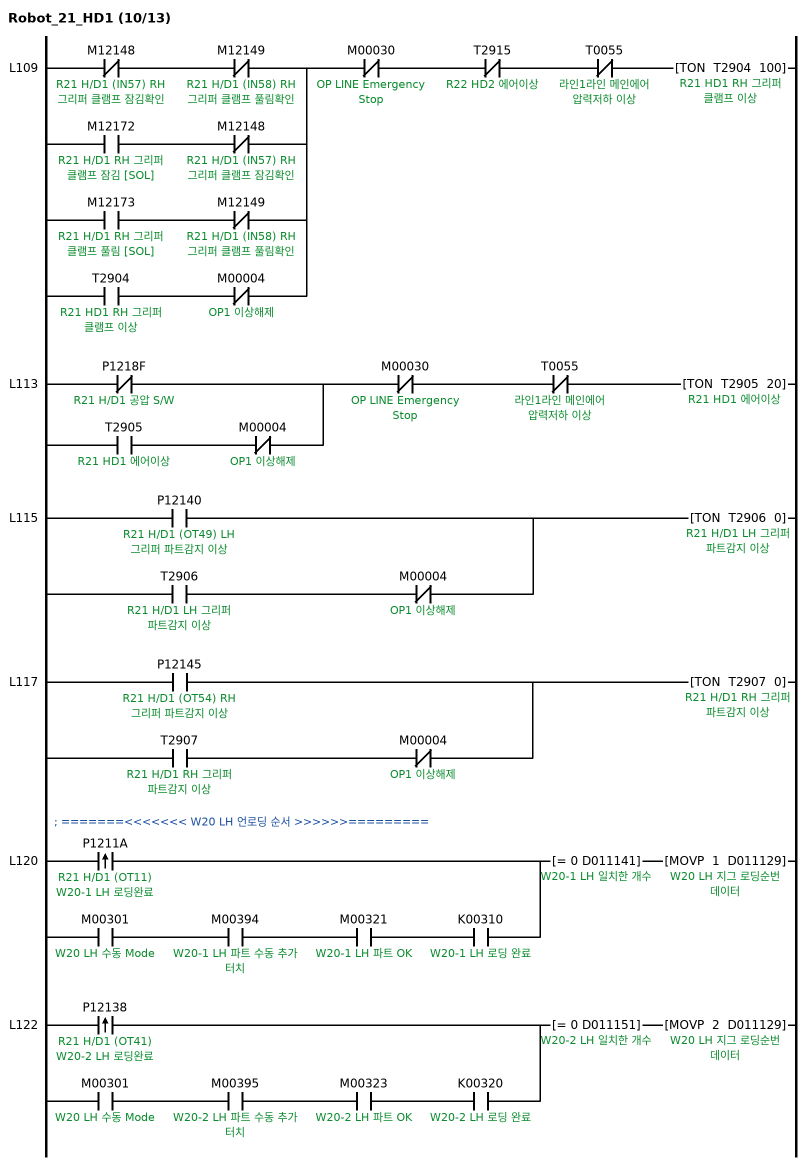
[picture p360: Robot_21_HD1 rungs L109-L122]
; L109
LOAD NOT  M12148	// R21 H/D1 (IN57) RH 그리퍼 클램프 잠김확인
AND NOT   M12149	// R21 H/D1 (IN58) RH 그리퍼 클램프 풀림확인
LOAD      M12172	// R21 H/D1 RH 그리퍼 클램프 잠김 [SOL]
AND NOT   M12148	// R21 H/D1 (IN57) RH 그리퍼 클램프 잠김확인
OR LOAD
LOAD      M12173	// R21 H/D1 RH 그리퍼 클램프 풀림 [SOL]
AND NOT   M12149	// R21 H/D1 (IN58) RH 그리퍼 클램프 풀림확인
OR LOAD
LOAD      T2904	// R21 HD1 RH 그리퍼 클램프 이상
AND NOT   M00004	// OP1 이상해제
OR LOAD
AND NOT   M00030	// OP LINE Emergency Stop
AND NOT   T2915	// R22 HD2 에어이상
AND NOT   T0055	// 라인1라인 메인에어 압력저하 이상
TON       T2904 100	// R21 HD1 RH 그리퍼 클램프 이상
; L113
LOAD NOT  P1218F	// R21 H/D1 공압 S/W
LOAD      T2905	// R21 HD1 에어이상
AND NOT   M00004	// OP1 이상해제
OR LOAD
AND NOT   M00030	// OP LINE Emergency Stop
AND NOT   T0055	// 라인1라인 메인에어 압력저하 이상
TON       T2905 20	// R21 HD1 에어이상
; L115
LOAD      P12140	// R21 H/D1 (OT49) LH 그리퍼 파트감지 이상
LOAD      T2906	// R21 H/D1 LH 그리퍼 파트감지 이상
AND NOT   M00004	// OP1 이상해제
OR LOAD
TON       T2906 0	// R21 H/D1 LH 그리퍼 파트감지 이상
; L117
LOAD      P12145	// R21 H/D1 (OT54) RH 그리퍼 파트감지 이상
LOAD      T2907	// R21 H/D1 RH 그리퍼 파트감지 이상
AND NOT   M00004	// OP1 이상해제
OR LOAD
TON       T2907 0	// R21 H/D1 RH 그리퍼 파트감지 이상
// =======<<<<<<< W20 LH 언로딩 순서 >>>>>>=========
; L120
LOADP     P1211A	// R21 H/D1 (OT11) W20-1 LH 로딩완료
LOAD      M00301	// W20 LH 수동 Mode
AND       M00394	// W20-1 LH 파트 수동 추가 터치
AND       M00321	// W20-1 LH 파트 OK
AND       K00310	// W20-1 LH 로딩 완료
OR LOAD
AND=      0 D011141	// W20-1 LH 일치한 개수
MOVP      1 D011129	// W20 LH 지그 로딩순번 데이터
; L122
LOADP     P12138	// R21 H/D1 (OT41) W20-2 LH 로딩완료
LOAD      M00301	// W20 LH 수동 Mode
AND       M00395	// W20-2 LH 파트 수동 추가 터치
AND       M00323	// W20-2 LH 파트 OK
AND       K00320	// W20-2 LH 로딩 완료
OR LOAD
AND=      0 D011151	// W20-2 LH 일치한 개수
MOVP      2 D011129	// W20 LH 지그 로딩순번 데이터

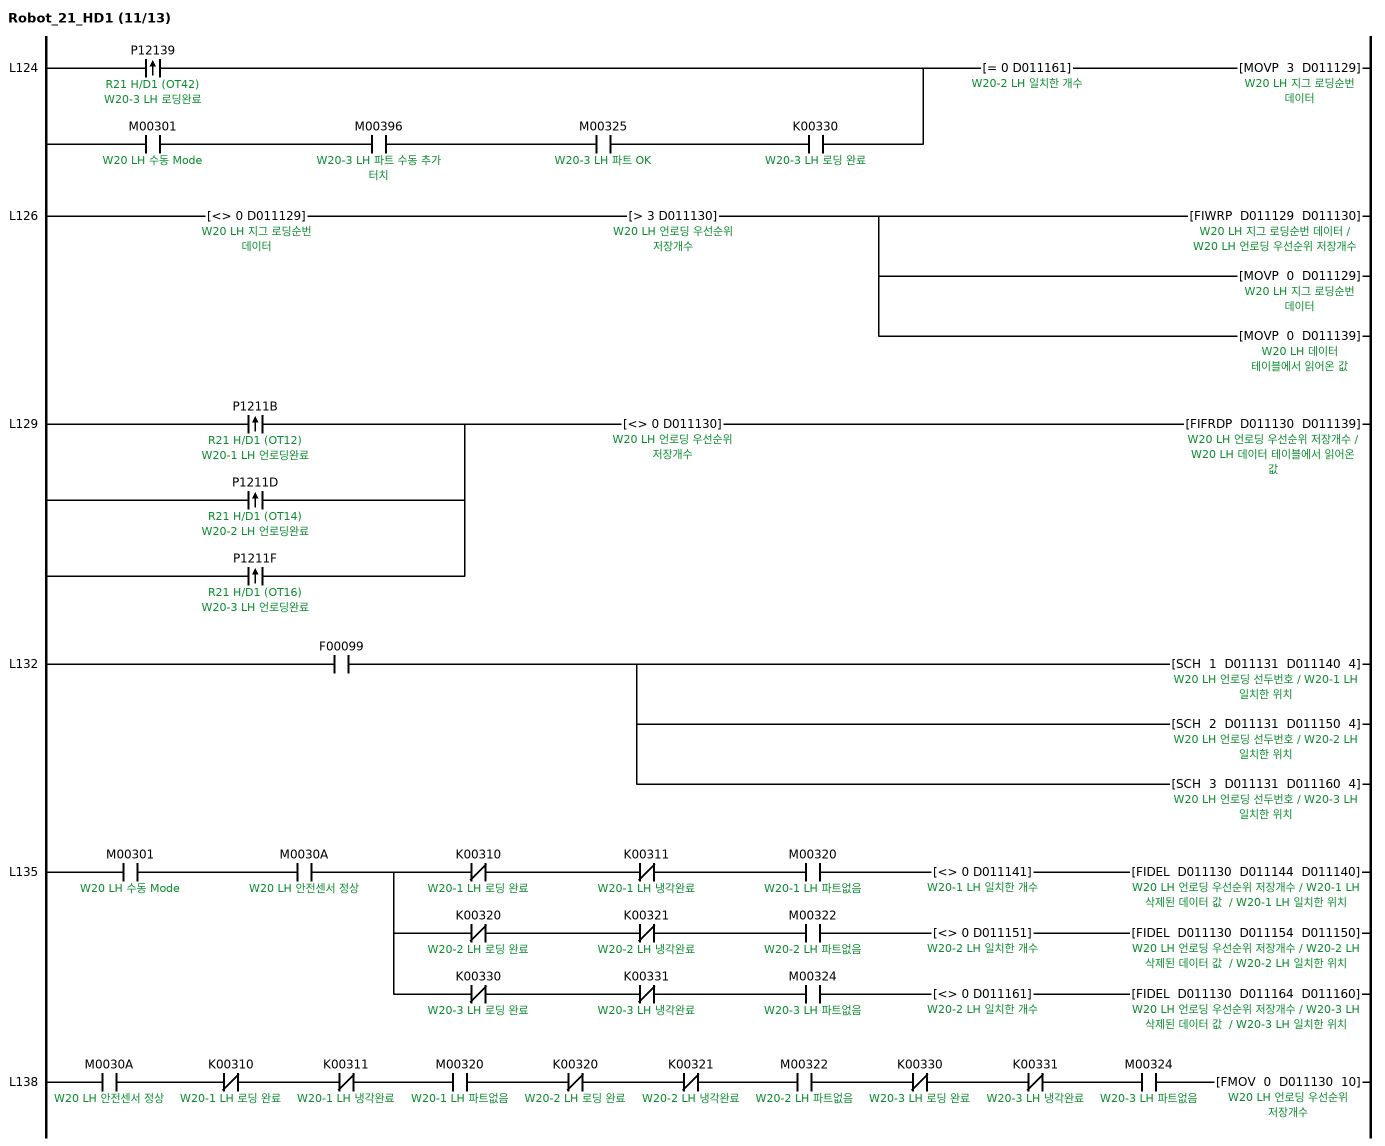
; L124
LOADP     P12139	// R21 H/D1 (OT42) W20-3 LH 로딩완료
LOAD      M00301	// W20 LH 수동 Mode
AND       M00396	// W20-3 LH 파트 수동 추가 터치
AND       M00325	// W20-3 LH 파트 OK
AND       K00330	// W20-3 LH 로딩 완료
OR LOAD
AND=      0 D011161	// W20-2 LH 일치한 개수
MOVP      3 D011129	// W20 LH 지그 로딩순번 데이터
; L126
LOAD<>    0 D011129	// W20 LH 지그 로딩순번 데이터
AND>      3 D011130	// W20 LH 언로딩 우선순위 저장개수
FIWRP     D011129 D011130	// W20 LH 지그 로딩순번 데이터 / W20 LH 언로딩 우선순위 저장개수
MOVP      0 D011129	// W20 LH 지그 로딩순번 데이터
MOVP      0 D011139	// W20 LH 데이터 테이블에서 읽어온 값
; L129
LOADP     P1211B	// R21 H/D1 (OT12) W20-1 LH 언로딩완료
ORP       P1211D	// R21 H/D1 (OT14) W20-2 LH 언로딩완료
ORP       P1211F	// R21 H/D1 (OT16) W20-3 LH 언로딩완료
AND<>     0 D011130	// W20 LH 언로딩 우선순위 저장개수
FIFRDP    D011130 D011139	// W20 LH 언로딩 우선순위 저장개수 / W20 LH 데이터 테이블에서 읽어온 값
; L132
LOAD      F00099
SCH       1 D011131 D011140 4	// W20 LH 언로딩 선두번호 / W20-1 LH 일치한 위치
SCH       2 D011131 D011150 4	// W20 LH 언로딩 선두번호 / W20-2 LH 일치한 위치
SCH       3 D011131 D011160 4	// W20 LH 언로딩 선두번호 / W20-3 LH 일치한 위치
; L135
LOAD      M00301	// W20 LH 수동 Mode
AND       M0030A	// W20 LH 안전센서 정상
MPUSH
AND NOT   K00310	// W20-1 LH 로딩 완료
AND NOT   K00311	// W20-1 LH 냉각완료
AND       M00320	// W20-1 LH 파트없음
AND<>     0 D011141	// W20-1 LH 일치한 개수
FIDEL     D011130 D011144 D011140	// W20 LH 언로딩 우선순위 저장개수 / W20-1 LH 삭제된 데이터 값  / W20-1 LH 일치한 위치
MLOAD
AND NOT   K00320	// W20-2 LH 로딩 완료
AND NOT   K00321	// W20-2 LH 냉각완료
AND       M00322	// W20-2 LH 파트없음
AND<>     0 D011151	// W20-2 LH 일치한 개수
FIDEL     D011130 D011154 D011150	// W20 LH 언로딩 우선순위 저장개수 / W20-2 LH 삭제된 데이터 값  / W20-2 LH 일치한 위치
MPOP
AND NOT   K00330	// W20-3 LH 로딩 완료
AND NOT   K00331	// W20-3 LH 냉각완료
AND       M00324	// W20-3 LH 파트없음
AND<>     0 D011161	// W20-2 LH 일치한 개수
FIDEL     D011130 D011164 D011160	// W20 LH 언로딩 우선순위 저장개수 / W20-3 LH 삭제된 데이터 값  / W20-3 LH 일치한 위치
; L138
LOAD      M0030A	// W20 LH 안전센서 정상
AND NOT   K00310	// W20-1 LH 로딩 완료
AND NOT   K00311	// W20-1 LH 냉각완료
AND       M00320	// W20-1 LH 파트없음
AND NOT   K00320	// W20-2 LH 로딩 완료
AND NOT   K00321	// W20-2 LH 냉각완료
AND       M00322	// W20-2 LH 파트없음
AND NOT   K00330	// W20-3 LH 로딩 완료
AND NOT   K00331	// W20-3 LH 냉각완료
AND       M00324	// W20-3 LH 파트없음
FMOV      0 D011130 10	// W20 LH 언로딩 우선순위 저장개수

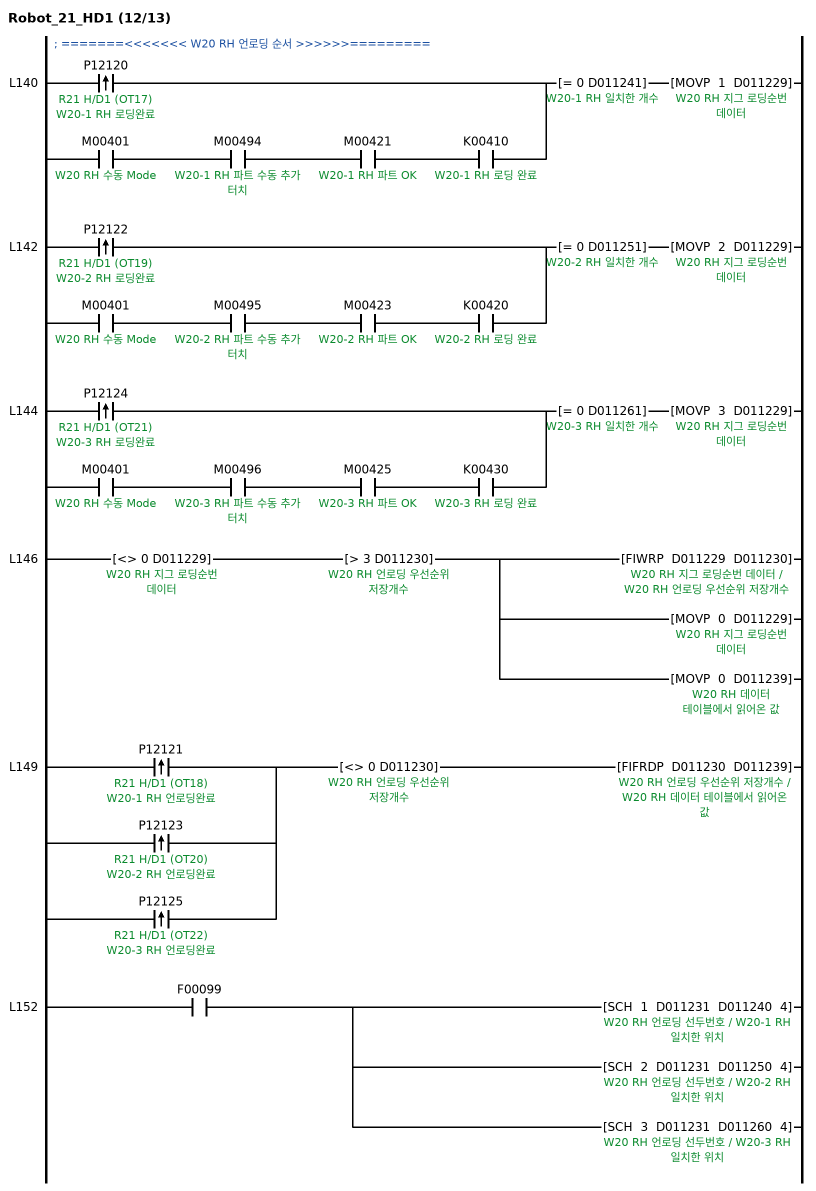
// =======<<<<<<< W20 RH 언로딩 순서 >>>>>>=========
; L140
LOADP     P12120	// R21 H/D1 (OT17) W20-1 RH 로딩완료
LOAD      M00401	// W20 RH 수동 Mode
AND       M00494	// W20-1 RH 파트 수동 추가 터치
AND       M00421	// W20-1 RH 파트 OK
AND       K00410	// W20-1 RH 로딩 완료
OR LOAD
AND=      0 D011241	// W20-1 RH 일치한 개수
MOVP      1 D011229	// W20 RH 지그 로딩순번 데이터
; L142
LOADP     P12122	// R21 H/D1 (OT19) W20-2 RH 로딩완료
LOAD      M00401	// W20 RH 수동 Mode
AND       M00495	// W20-2 RH 파트 수동 추가 터치
AND       M00423	// W20-2 RH 파트 OK
AND       K00420	// W20-2 RH 로딩 완료
OR LOAD
AND=      0 D011251	// W20-2 RH 일치한 개수
MOVP      2 D011229	// W20 RH 지그 로딩순번 데이터
; L144
LOADP     P12124	// R21 H/D1 (OT21) W20-3 RH 로딩완료
LOAD      M00401	// W20 RH 수동 Mode
AND       M00496	// W20-3 RH 파트 수동 추가 터치
AND       M00425	// W20-3 RH 파트 OK
AND       K00430	// W20-3 RH 로딩 완료
OR LOAD
AND=      0 D011261	// W20-3 RH 일치한 개수
MOVP      3 D011229	// W20 RH 지그 로딩순번 데이터
; L146
LOAD<>    0 D011229	// W20 RH 지그 로딩순번 데이터
AND>      3 D011230	// W20 RH 언로딩 우선순위 저장개수
FIWRP     D011229 D011230	// W20 RH 지그 로딩순번 데이터 / W20 RH 언로딩 우선순위 저장개수
MOVP      0 D011229	// W20 RH 지그 로딩순번 데이터
MOVP      0 D011239	// W20 RH 데이터 테이블에서 읽어온 값
; L149
LOADP     P12121	// R21 H/D1 (OT18) W20-1 RH 언로딩완료
ORP       P12123	// R21 H/D1 (OT20) W20-2 RH 언로딩완료
ORP       P12125	// R21 H/D1 (OT22) W20-3 RH 언로딩완료
AND<>     0 D011230	// W20 RH 언로딩 우선순위 저장개수
FIFRDP    D011230 D011239	// W20 RH 언로딩 우선순위 저장개수 / W20 RH 데이터 테이블에서 읽어온 값
; L152
LOAD      F00099
SCH       1 D011231 D011240 4	// W20 RH 언로딩 선두번호 / W20-1 RH 일치한 위치
SCH       2 D011231 D011250 4	// W20 RH 언로딩 선두번호 / W20-2 RH 일치한 위치
SCH       3 D011231 D011260 4	// W20 RH 언로딩 선두번호 / W20-3 RH 일치한 위치

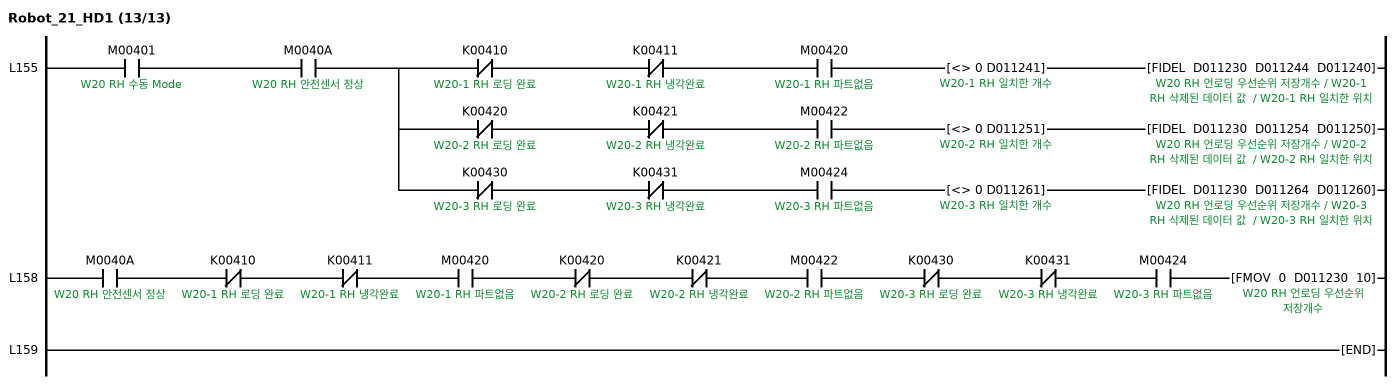
; L155
LOAD      M00401	// W20 RH 수동 Mode
AND       M0040A	// W20 RH 안전센서 정상
MPUSH
AND NOT   K00410	// W20-1 RH 로딩 완료
AND NOT   K00411	// W20-1 RH 냉각완료
AND       M00420	// W20-1 RH 파트없음
AND<>     0 D011241	// W20-1 RH 일치한 개수
FIDEL     D011230 D011244 D011240	// W20 RH 언로딩 우선순위 저장개수 / W20-1 RH 삭제된 데이터 값  / W20-1 RH 일치한 위치
MLOAD
AND NOT   K00420	// W20-2 RH 로딩 완료
AND NOT   K00421	// W20-2 RH 냉각완료
AND       M00422	// W20-2 RH 파트없음
AND<>     0 D011251	// W20-2 RH 일치한 개수
FIDEL     D011230 D011254 D011250	// W20 RH 언로딩 우선순위 저장개수 / W20-2 RH 삭제된 데이터 값  / W20-2 RH 일치한 위치
MPOP
AND NOT   K00430	// W20-3 RH 로딩 완료
AND NOT   K00431	// W20-3 RH 냉각완료
AND       M00424	// W20-3 RH 파트없음
AND<>     0 D011261	// W20-3 RH 일치한 개수
FIDEL     D011230 D011264 D011260	// W20 RH 언로딩 우선순위 저장개수 / W20-3 RH 삭제된 데이터 값  / W20-3 RH 일치한 위치
; L158
LOAD      M0040A	// W20 RH 안전센서 정상
AND NOT   K00410	// W20-1 RH 로딩 완료
AND NOT   K00411	// W20-1 RH 냉각완료
AND       M00420	// W20-1 RH 파트없음
AND NOT   K00420	// W20-2 RH 로딩 완료
AND NOT   K00421	// W20-2 RH 냉각완료
AND       M00422	// W20-2 RH 파트없음
AND NOT   K00430	// W20-3 RH 로딩 완료
AND NOT   K00431	// W20-3 RH 냉각완료
AND       M00424	// W20-3 RH 파트없음
FMOV      0 D011230 10	// W20 RH 언로딩 우선순위 저장개수
; L159
END

PROGRAM Robot_22_HD2 (task: 스캔 프로그램)

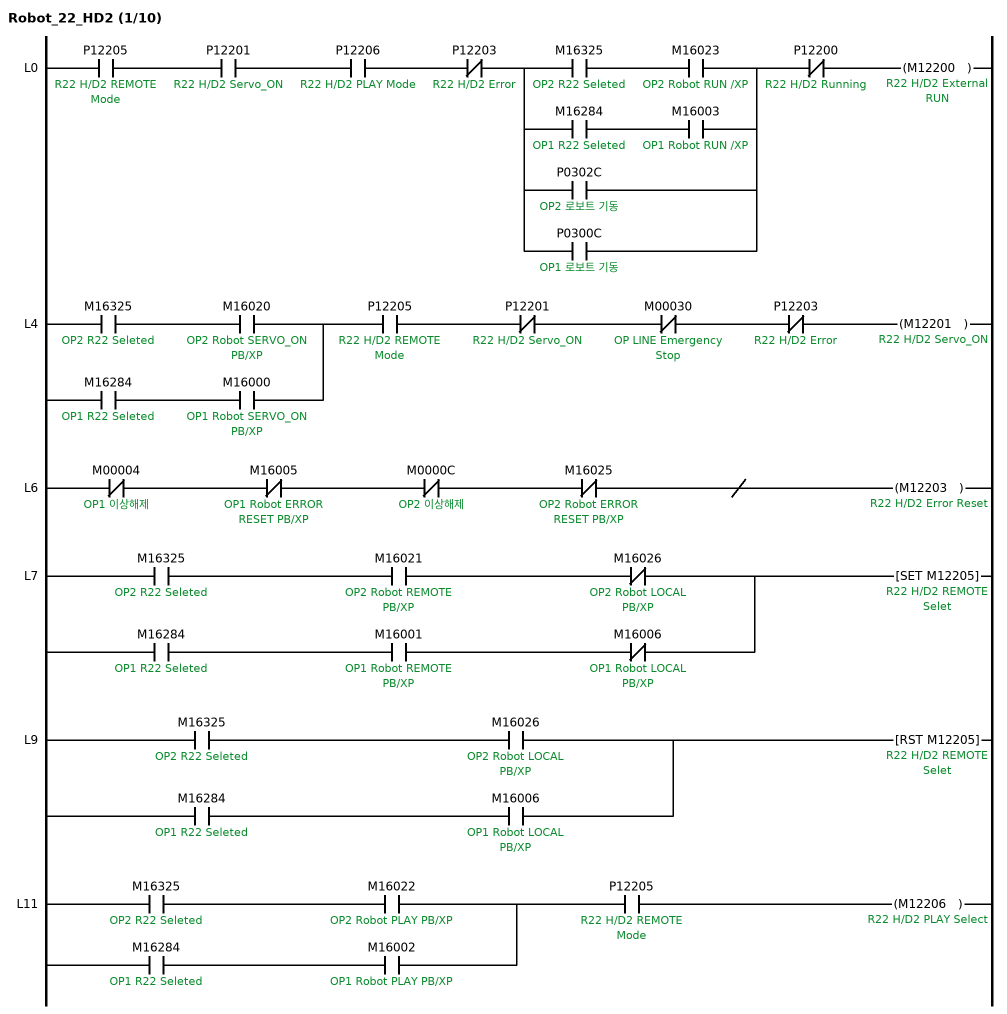
; L0
LOAD      P12205	// R22 H/D2 REMOTE Mode
AND       P12201	// R22 H/D2 Servo_ON
AND       P12206	// R22 H/D2 PLAY Mode
AND NOT   P12203	// R22 H/D2 Error
LOAD      M16325	// OP2 R22 Seleted
AND       M16023	// OP2 Robot RUN /XP
LOAD      M16284	// OP1 R22 Seleted
AND       M16003	// OP1 Robot RUN /XP
OR LOAD
OR        P0302C	// OP2 로보트 기동
OR        P0300C	// OP1 로보트 기동
AND LOAD
AND NOT   P12200	// R22 H/D2 Running
OUT       M12200	// R22 H/D2 External RUN
; L4
LOAD      M16325	// OP2 R22 Seleted
AND       M16020	// OP2 Robot SERVO_ON PB/XP
LOAD      M16284	// OP1 R22 Seleted
AND       M16000	// OP1 Robot SERVO_ON PB/XP
OR LOAD
AND       P12205	// R22 H/D2 REMOTE Mode
AND NOT   P12201	// R22 H/D2 Servo_ON
AND NOT   M00030	// OP LINE Emergency Stop
AND NOT   P12203	// R22 H/D2 Error
OUT       M12201	// R22 H/D2 Servo_ON
; L6
LOAD NOT  M00004	// OP1 이상해제
AND NOT   M16005	// OP1 Robot ERROR RESET PB/XP
AND NOT   M0000C	// OP2 이상해제
AND NOT   M16025	// OP2 Robot ERROR RESET PB/XP
NOT
OUT       M12203	// R22 H/D2 Error Reset
; L7
LOAD      M16325	// OP2 R22 Seleted
AND       M16021	// OP2 Robot REMOTE PB/XP
AND NOT   M16026	// OP2 Robot LOCAL PB/XP
LOAD      M16284	// OP1 R22 Seleted
AND       M16001	// OP1 Robot REMOTE PB/XP
AND NOT   M16006	// OP1 Robot LOCAL PB/XP
OR LOAD
SET       M12205	// R22 H/D2 REMOTE Selet
; L9
LOAD      M16325	// OP2 R22 Seleted
AND       M16026	// OP2 Robot LOCAL PB/XP
LOAD      M16284	// OP1 R22 Seleted
AND       M16006	// OP1 Robot LOCAL PB/XP
OR LOAD
RST       M12205	// R22 H/D2 REMOTE Selet
; L11
LOAD      M16325	// OP2 R22 Seleted
AND       M16022	// OP2 Robot PLAY PB/XP
LOAD      M16284	// OP1 R22 Seleted
AND       M16002	// OP1 Robot PLAY PB/XP
OR LOAD
AND       P12205	// R22 H/D2 REMOTE Mode
OUT       M12206	// R22 H/D2 PLAY Select

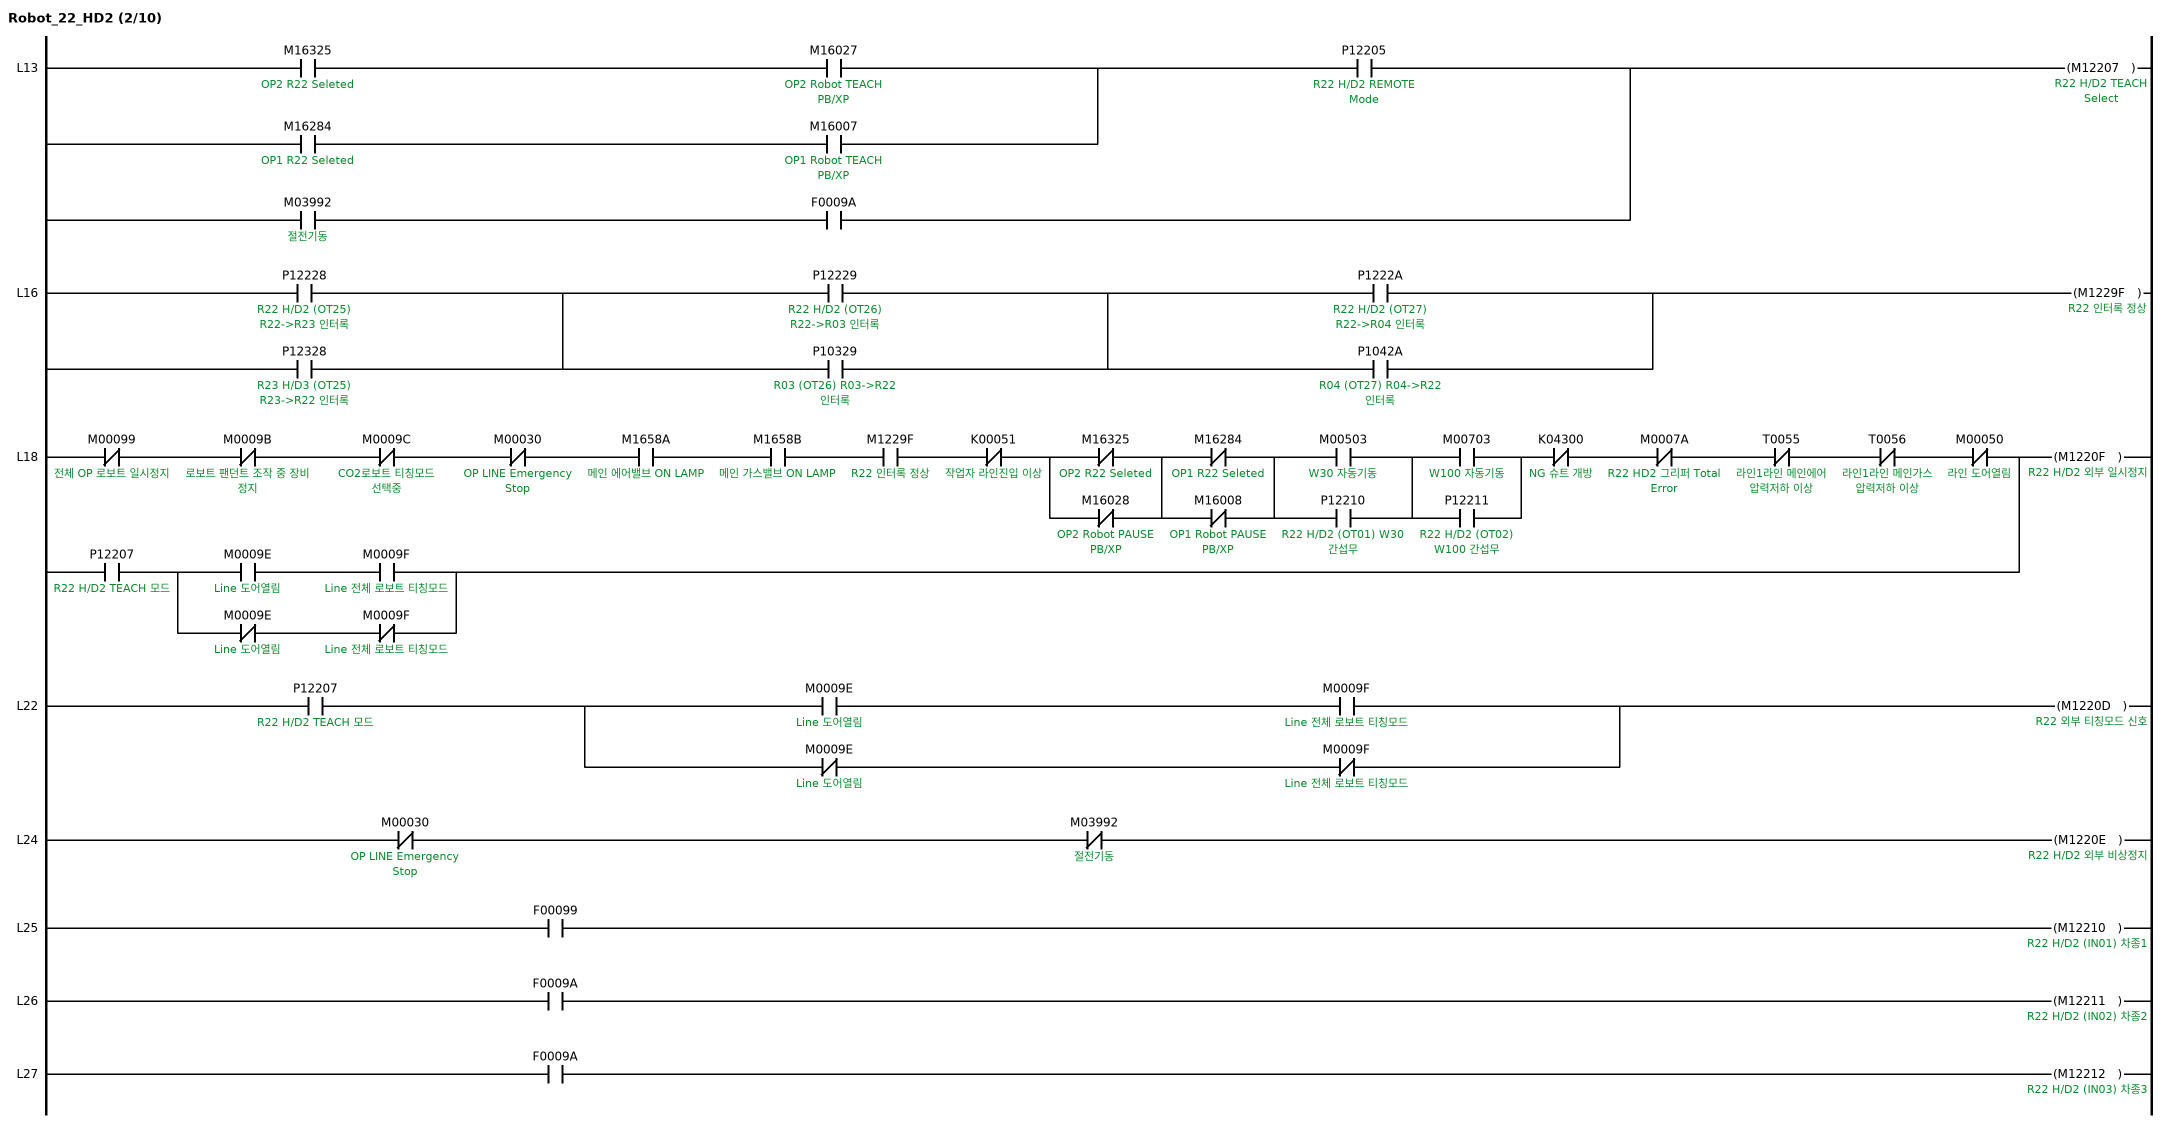
; L13
LOAD      M16325	// OP2 R22 Seleted
AND       M16027	// OP2 Robot TEACH PB/XP
LOAD      M16284	// OP1 R22 Seleted
AND       M16007	// OP1 Robot TEACH PB/XP
OR LOAD
AND       P12205	// R22 H/D2 REMOTE Mode
LOAD      M03992	// 절전기동
AND       F0009A
OR LOAD
OUT       M12207	// R22 H/D2 TEACH Select
; L16
LOAD      P12228	// R22 H/D2 (OT25) R22->R23 인터록
OR        P12328	// R23 H/D3 (OT25) R23->R22 인터록
LOAD      P12229	// R22 H/D2 (OT26) R22->R03 인터록
OR        P10329	// R03 (OT26) R03->R22 인터록
AND LOAD
LOAD      P1222A	// R22 H/D2 (OT27) R22->R04 인터록
OR        P1042A	// R04 (OT27) R04->R22 인터록
AND LOAD
OUT       M1229F	// R22 인터록 정상
; L18
LOAD NOT  M00099	// 전체 OP 로보트 일시정지
AND NOT   M0009B	// 로보트 팬던트 조작 중 장비 정지
AND NOT   M0009C	// CO2로보트 티칭모드 선택중
AND NOT   M00030	// OP LINE Emergency Stop
AND       M1658A	// 메인 에어밸브 ON LAMP
AND       M1658B	// 메인 가스밸브 ON LAMP
AND       M1229F	// R22 인터록 정상
AND NOT   K00051	//  작업자 라인진입 이상
LOAD NOT  M16325	// OP2 R22 Seleted
OR NOT    M16028	// OP2 Robot PAUSE PB/XP
AND LOAD
LOAD NOT  M16284	// OP1 R22 Seleted
OR NOT    M16008	// OP1 Robot PAUSE PB/XP
AND LOAD
LOAD      M00503	// W30 자동기동
OR        P12210	// R22 H/D2 (OT01) W30 간섭무
AND LOAD
LOAD      M00703	// W100 자동기동
OR        P12211	// R22 H/D2 (OT02) W100 간섭무
AND LOAD
AND NOT   K04300	// NG 슈트 개방
AND NOT   M0007A	// R22 HD2 그리퍼 Total Error 
AND NOT   T0055	// 라인1라인 메인에어 압력저하 이상
AND NOT   T0056	// 라인1라인 메인가스 압력저하 이상
AND NOT   M00050	// 라인 도어열림
LOAD      P12207	// R22 H/D2 TEACH 모드
LOAD      M0009E	// Line 도어열림
AND       M0009F	// Line 전체 로보트 티칭모드
LOAD NOT  M0009E	// Line 도어열림
AND NOT   M0009F	// Line 전체 로보트 티칭모드
OR LOAD
AND LOAD
OR LOAD
OUT       M1220F	// R22 H/D2 외부 일시정지
; L22
LOAD      P12207	// R22 H/D2 TEACH 모드
LOAD      M0009E	// Line 도어열림
AND       M0009F	// Line 전체 로보트 티칭모드
LOAD NOT  M0009E	// Line 도어열림
AND NOT   M0009F	// Line 전체 로보트 티칭모드
OR LOAD
AND LOAD
OUT       M1220D	// R22 외부 티칭모드 신호
; L24
LOAD NOT  M00030	// OP LINE Emergency Stop
AND NOT   M03992	// 절전기동
OUT       M1220E	// R22 H/D2 외부 비상정지 
; L25
LOAD      F00099
OUT       M12210	// R22 H/D2 (IN01) 차종1
; L26
LOAD      F0009A
OUT       M12211	// R22 H/D2 (IN02) 차종2
; L27
LOAD      F0009A
OUT       M12212	// R22 H/D2 (IN03) 차종3

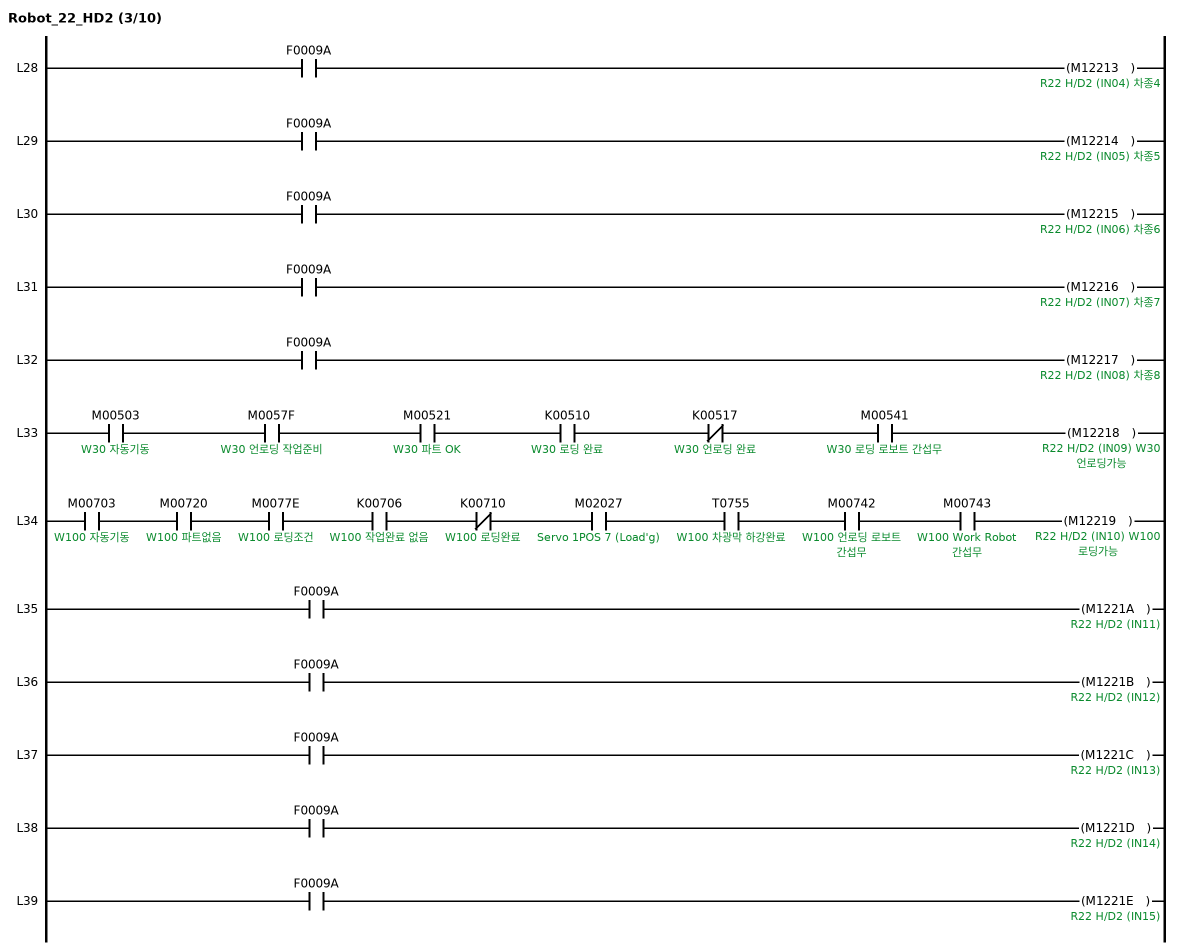
; L28
LOAD      F0009A
OUT       M12213	// R22 H/D2 (IN04) 차종4
; L29
LOAD      F0009A
OUT       M12214	// R22 H/D2 (IN05) 차종5
; L30
LOAD      F0009A
OUT       M12215	// R22 H/D2 (IN06) 차종6
; L31
LOAD      F0009A
OUT       M12216	// R22 H/D2 (IN07) 차종7
; L32
LOAD      F0009A
OUT       M12217	// R22 H/D2 (IN08) 차종8
; L33
LOAD      M00503	// W30 자동기동
AND       M0057F	// W30 언로딩 작업준비
AND       M00521	// W30 파트 OK
AND       K00510	// W30 로딩 완료
AND NOT   K00517	// W30 언로딩 완료
AND       M00541	// W30 로딩 로보트 간섭무
OUT       M12218	// R22 H/D2 (IN09) W30 언로딩가능
; L34
LOAD      M00703	// W100 자동기동
AND       M00720	// W100 파트없음
AND       M0077E	// W100 로딩조건
AND       K00706	// W100 작업완료 없음
AND NOT   K00710	// W100 로딩완료
AND       M02027	// Servo 1POS 7 (Load'g)
AND       T0755	// W100 차광막 하강완료
AND       M00742	// W100 언로딩 로보트 간섭무
AND       M00743	// W100 Work Robot 간섭무
OUT       M12219	// R22 H/D2 (IN10) W100 로딩가능
; L35
LOAD      F0009A
OUT       M1221A	// R22 H/D2 (IN11)
; L36
LOAD      F0009A
OUT       M1221B	// R22 H/D2 (IN12)
; L37
LOAD      F0009A
OUT       M1221C	// R22 H/D2 (IN13)
; L38
LOAD      F0009A
OUT       M1221D	// R22 H/D2 (IN14)
; L39
LOAD      F0009A
OUT       M1221E	// R22 H/D2 (IN15)

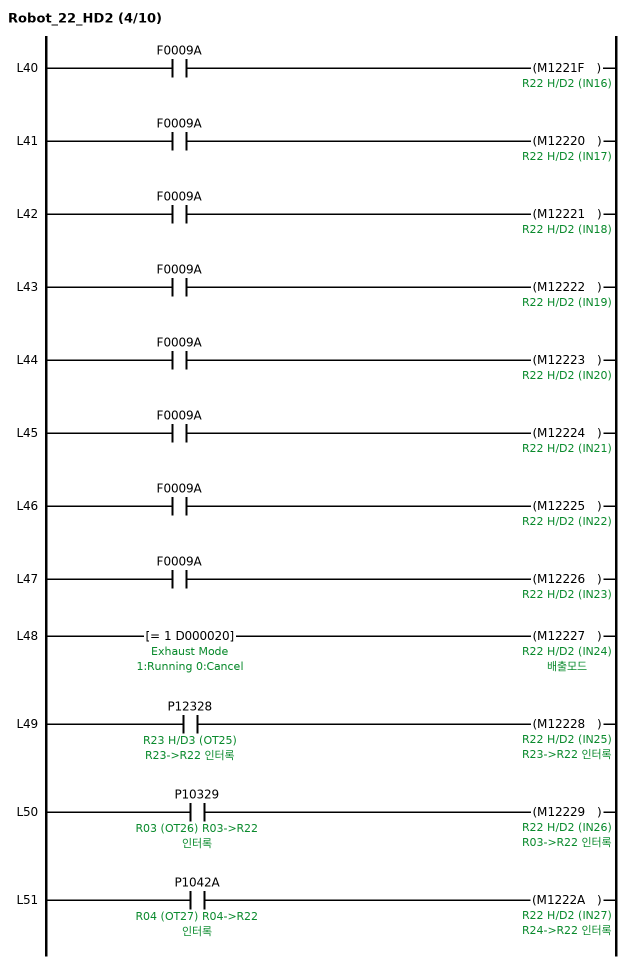
; L40
LOAD      F0009A
OUT       M1221F	// R22 H/D2 (IN16)
; L41
LOAD      F0009A
OUT       M12220	// R22 H/D2 (IN17)
; L42
LOAD      F0009A
OUT       M12221	// R22 H/D2 (IN18)
; L43
LOAD      F0009A
OUT       M12222	// R22 H/D2 (IN19)
; L44
LOAD      F0009A
OUT       M12223	// R22 H/D2 (IN20)
; L45
LOAD      F0009A
OUT       M12224	// R22 H/D2 (IN21)
; L46
LOAD      F0009A
OUT       M12225	// R22 H/D2 (IN22)
; L47
LOAD      F0009A
OUT       M12226	// R22 H/D2 (IN23)
; L48
LOAD=     1 D000020	// Exhaust Mode 1:Running 0:Cancel
OUT       M12227	// R22 H/D2 (IN24) 배출모드
; L49
LOAD      P12328	// R23 H/D3 (OT25) R23->R22 인터록
OUT       M12228	// R22 H/D2 (IN25) R23->R22 인터록
; L50
LOAD      P10329	// R03 (OT26) R03->R22 인터록
OUT       M12229	// R22 H/D2 (IN26) R03->R22 인터록
; L51
LOAD      P1042A	// R04 (OT27) R04->R22 인터록
OUT       M1222A	// R22 H/D2 (IN27) R24->R22 인터록

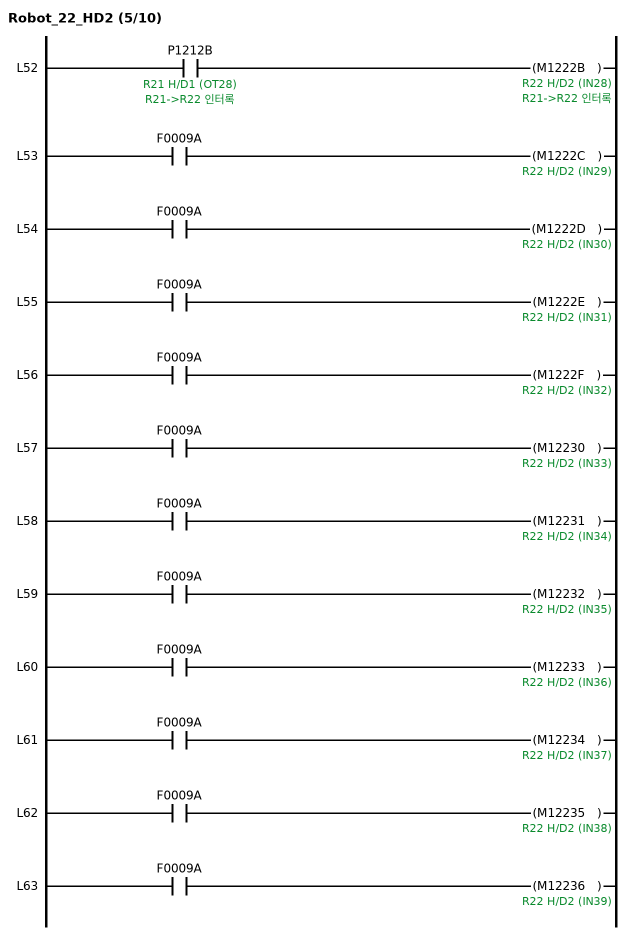
; L52
LOAD      P1212B	// R21 H/D1 (OT28) R21->R22 인터록
OUT       M1222B	// R22 H/D2 (IN28) R21->R22 인터록
; L53
LOAD      F0009A
OUT       M1222C	// R22 H/D2 (IN29)
; L54
LOAD      F0009A
OUT       M1222D	// R22 H/D2 (IN30)
; L55
LOAD      F0009A
OUT       M1222E	// R22 H/D2 (IN31)
; L56
LOAD      F0009A
OUT       M1222F	// R22 H/D2 (IN32)
; L57
LOAD      F0009A
OUT       M12230	// R22 H/D2 (IN33)
; L58
LOAD      F0009A
OUT       M12231	// R22 H/D2 (IN34)
; L59
LOAD      F0009A
OUT       M12232	// R22 H/D2 (IN35)
; L60
LOAD      F0009A
OUT       M12233	// R22 H/D2 (IN36)
; L61
LOAD      F0009A
OUT       M12234	// R22 H/D2 (IN37)
; L62
LOAD      F0009A
OUT       M12235	// R22 H/D2 (IN38)
; L63
LOAD      F0009A
OUT       M12236	// R22 H/D2 (IN39)

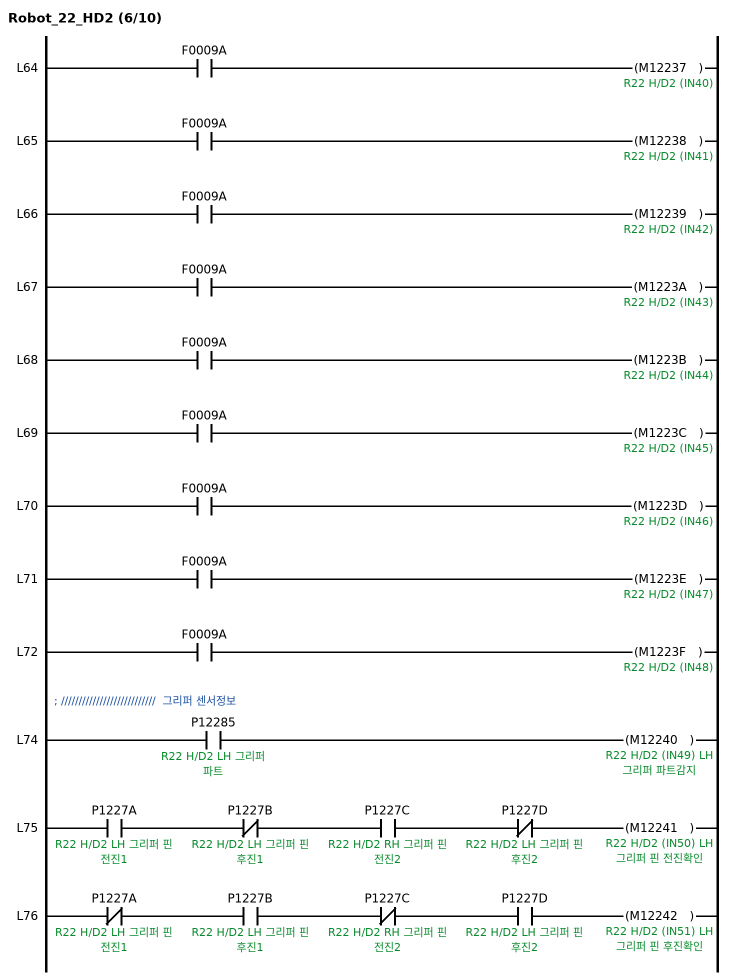
; L64
LOAD      F0009A
OUT       M12237	// R22 H/D2 (IN40)
; L65
LOAD      F0009A
OUT       M12238	// R22 H/D2 (IN41)
; L66
LOAD      F0009A
OUT       M12239	// R22 H/D2 (IN42)
; L67
LOAD      F0009A
OUT       M1223A	// R22 H/D2 (IN43)
; L68
LOAD      F0009A
OUT       M1223B	// R22 H/D2 (IN44)
; L69
LOAD      F0009A
OUT       M1223C	// R22 H/D2 (IN45)
; L70
LOAD      F0009A
OUT       M1223D	// R22 H/D2 (IN46)
; L71
LOAD      F0009A
OUT       M1223E	// R22 H/D2 (IN47)
; L72
LOAD      F0009A
OUT       M1223F	// R22 H/D2 (IN48)
// ///////////////////////////  그리퍼 센서정보
; L74
LOAD      P12285	// R22 H/D2 LH 그리퍼 파트
OUT       M12240	// R22 H/D2 (IN49) LH 그리퍼 파트감지
; L75
LOAD      P1227A	// R22 H/D2 LH 그리퍼 핀 전진1
AND NOT   P1227B	// R22 H/D2 LH 그리퍼 핀 후진1
AND       P1227C	// R22 H/D2 RH 그리퍼 핀 전진2
AND NOT   P1227D	// R22 H/D2 LH 그리퍼 핀 후진2
OUT       M12241	// R22 H/D2 (IN50) LH 그리퍼 핀 전진확인
; L76
LOAD NOT  P1227A	// R22 H/D2 LH 그리퍼 핀 전진1
AND       P1227B	// R22 H/D2 LH 그리퍼 핀 후진1
AND NOT   P1227C	// R22 H/D2 RH 그리퍼 핀 전진2
AND       P1227D	// R22 H/D2 LH 그리퍼 핀 후진2
OUT       M12242	// R22 H/D2 (IN51) LH 그리퍼 핀 후진확인

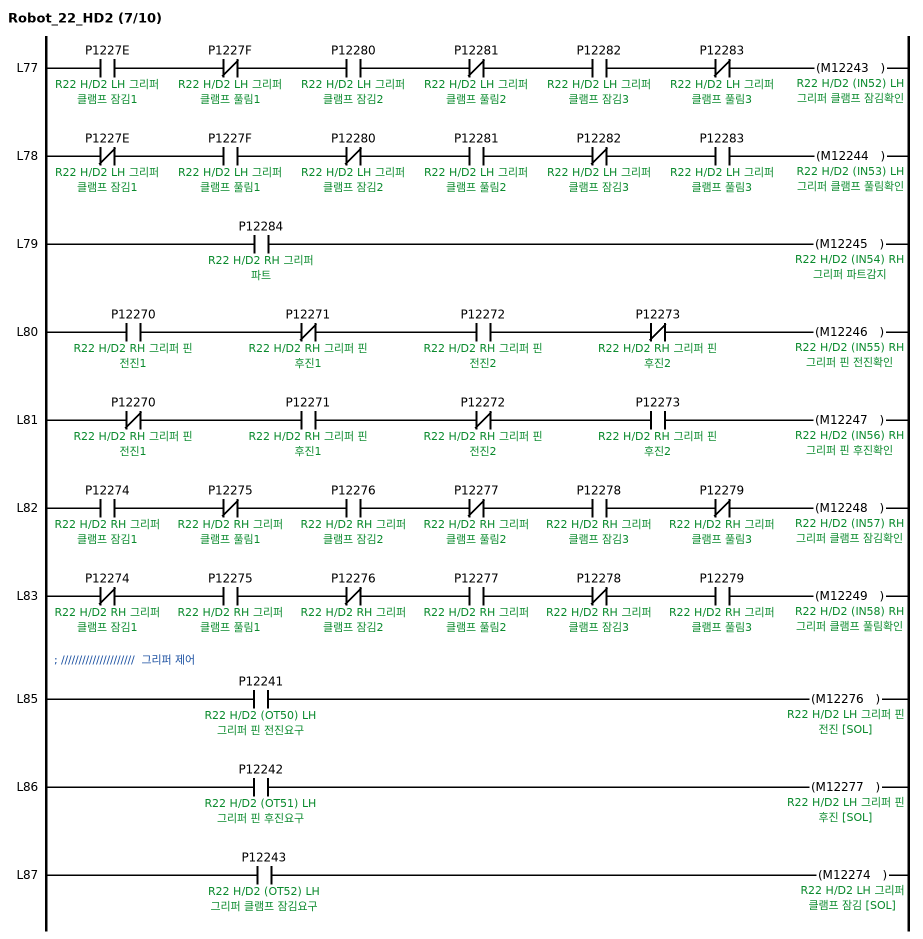
; L77
LOAD      P1227E	// R22 H/D2 LH 그리퍼 클램프 잠김1
AND NOT   P1227F	// R22 H/D2 LH 그리퍼 클램프 풀림1
AND       P12280	// R22 H/D2 LH 그리퍼 클램프 잠김2
AND NOT   P12281	// R22 H/D2 LH 그리퍼 클램프 풀림2
AND       P12282	// R22 H/D2 LH 그리퍼 클램프 잠김3
AND NOT   P12283	// R22 H/D2 LH 그리퍼 클램프 풀림3
OUT       M12243	// R22 H/D2 (IN52) LH 그리퍼 클램프 잠김확인
; L78
LOAD NOT  P1227E	// R22 H/D2 LH 그리퍼 클램프 잠김1
AND       P1227F	// R22 H/D2 LH 그리퍼 클램프 풀림1
AND NOT   P12280	// R22 H/D2 LH 그리퍼 클램프 잠김2
AND       P12281	// R22 H/D2 LH 그리퍼 클램프 풀림2
AND NOT   P12282	// R22 H/D2 LH 그리퍼 클램프 잠김3
AND       P12283	// R22 H/D2 LH 그리퍼 클램프 풀림3
OUT       M12244	// R22 H/D2 (IN53) LH 그리퍼 클램프 풀림확인
; L79
LOAD      P12284	// R22 H/D2 RH 그리퍼 파트
OUT       M12245	// R22 H/D2 (IN54) RH 그리퍼 파트감지
; L80
LOAD      P12270	// R22 H/D2 RH 그리퍼 핀 전진1
AND NOT   P12271	// R22 H/D2 RH 그리퍼 핀 후진1
AND       P12272	// R22 H/D2 RH 그리퍼 핀 전진2
AND NOT   P12273	// R22 H/D2 RH 그리퍼 핀 후진2
OUT       M12246	// R22 H/D2 (IN55) RH 그리퍼 핀 전진확인
; L81
LOAD NOT  P12270	// R22 H/D2 RH 그리퍼 핀 전진1
AND       P12271	// R22 H/D2 RH 그리퍼 핀 후진1
AND NOT   P12272	// R22 H/D2 RH 그리퍼 핀 전진2
AND       P12273	// R22 H/D2 RH 그리퍼 핀 후진2
OUT       M12247	// R22 H/D2 (IN56) RH 그리퍼 핀 후진확인
; L82
LOAD      P12274	// R22 H/D2 RH 그리퍼 클램프 잠김1
AND NOT   P12275	// R22 H/D2 RH 그리퍼 클램프 풀림1
AND       P12276	// R22 H/D2 RH 그리퍼 클램프 잠김2
AND NOT   P12277	// R22 H/D2 RH 그리퍼 클램프 풀림2
AND       P12278	// R22 H/D2 RH 그리퍼 클램프 잠김3
AND NOT   P12279	// R22 H/D2 RH 그리퍼 클램프 풀림3
OUT       M12248	// R22 H/D2 (IN57) RH 그리퍼 클램프 잠김확인
; L83
LOAD NOT  P12274	// R22 H/D2 RH 그리퍼 클램프 잠김1
AND       P12275	// R22 H/D2 RH 그리퍼 클램프 풀림1
AND NOT   P12276	// R22 H/D2 RH 그리퍼 클램프 잠김2
AND       P12277	// R22 H/D2 RH 그리퍼 클램프 풀림2
AND NOT   P12278	// R22 H/D2 RH 그리퍼 클램프 잠김3
AND       P12279	// R22 H/D2 RH 그리퍼 클램프 풀림3
OUT       M12249	// R22 H/D2 (IN58) RH 그리퍼 클램프 풀림확인
// /////////////////////  그리퍼 제어
; L85
LOAD      P12241	// R22 H/D2 (OT50) LH 그리퍼 핀 전진요구
OUT       M12276	// R22 H/D2 LH 그리퍼 핀 전진 [SOL]
; L86
LOAD      P12242	// R22 H/D2 (OT51) LH 그리퍼 핀 후진요구
OUT       M12277	// R22 H/D2 LH 그리퍼 핀 후진 [SOL]
; L87
LOAD      P12243	// R22 H/D2 (OT52) LH 그리퍼 클램프 잠김요구
OUT       M12274	// R22 H/D2 LH 그리퍼 클램프 잠김 [SOL]

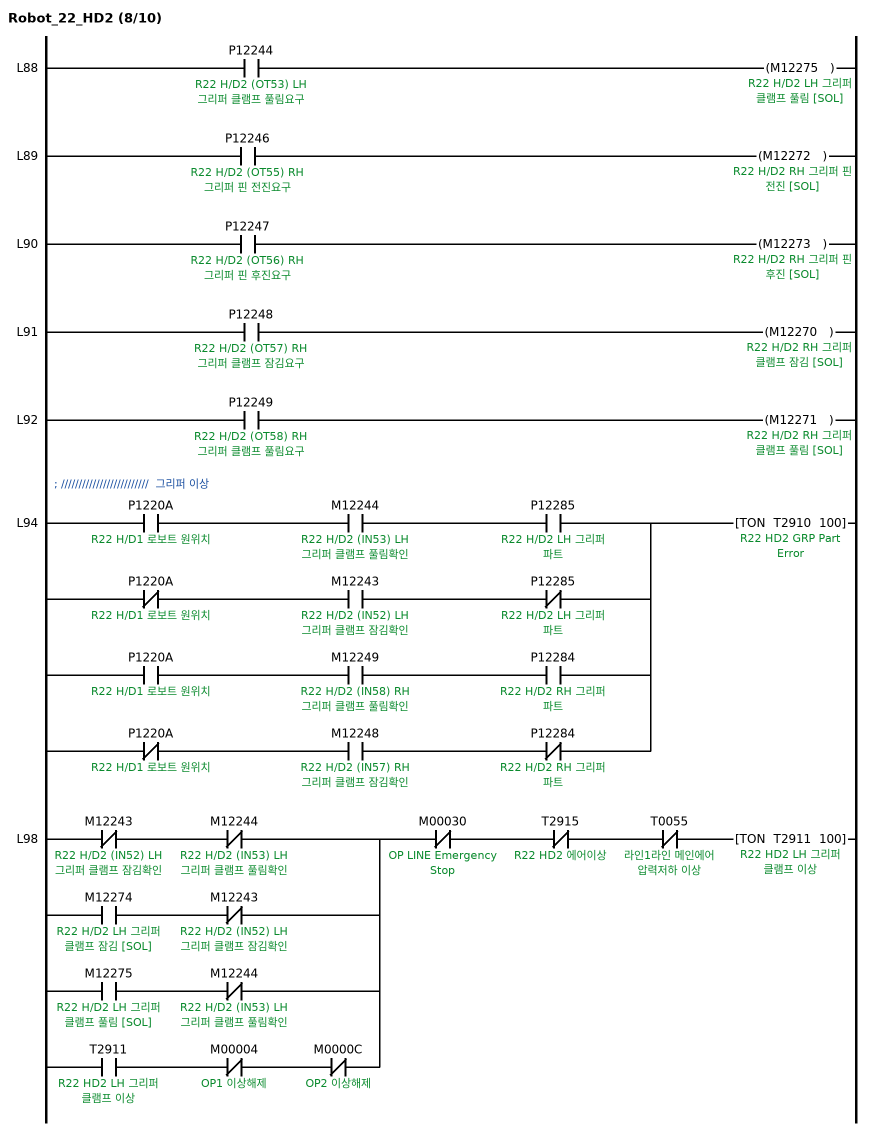
; L88
LOAD      P12244	// R22 H/D2 (OT53) LH 그리퍼 클램프 풀림요구
OUT       M12275	// R22 H/D2 LH 그리퍼 클램프 풀림 [SOL]
; L89
LOAD      P12246	// R22 H/D2 (OT55) RH 그리퍼 핀 전진요구
OUT       M12272	// R22 H/D2 RH 그리퍼 핀 전진 [SOL]
; L90
LOAD      P12247	// R22 H/D2 (OT56) RH 그리퍼 핀 후진요구
OUT       M12273	// R22 H/D2 RH 그리퍼 핀 후진 [SOL]
; L91
LOAD      P12248	// R22 H/D2 (OT57) RH 그리퍼 클램프 잠김요구
OUT       M12270	// R22 H/D2 RH 그리퍼 클램프 잠김 [SOL]
; L92
LOAD      P12249	// R22 H/D2 (OT58) RH 그리퍼 클램프 풀림요구
OUT       M12271	// R22 H/D2 RH 그리퍼 클램프 풀림 [SOL]
// /////////////////////////  그리퍼 이상
; L94
LOAD      P1220A	// R22 H/D1 로보트 원위치
AND       M12244	// R22 H/D2 (IN53) LH 그리퍼 클램프 풀림확인
AND       P12285	// R22 H/D2 LH 그리퍼 파트
LOAD NOT  P1220A	// R22 H/D1 로보트 원위치
AND       M12243	// R22 H/D2 (IN52) LH 그리퍼 클램프 잠김확인
AND NOT   P12285	// R22 H/D2 LH 그리퍼 파트
OR LOAD
LOAD      P1220A	// R22 H/D1 로보트 원위치
AND       M12249	// R22 H/D2 (IN58) RH 그리퍼 클램프 풀림확인
AND       P12284	// R22 H/D2 RH 그리퍼 파트
OR LOAD
LOAD NOT  P1220A	// R22 H/D1 로보트 원위치
AND       M12248	// R22 H/D2 (IN57) RH 그리퍼 클램프 잠김확인
AND NOT   P12284	// R22 H/D2 RH 그리퍼 파트
OR LOAD
TON       T2910 100	// R22 HD2 GRP Part Error 
; L98
LOAD NOT  M12243	// R22 H/D2 (IN52) LH 그리퍼 클램프 잠김확인
AND NOT   M12244	// R22 H/D2 (IN53) LH 그리퍼 클램프 풀림확인
LOAD      M12274	// R22 H/D2 LH 그리퍼 클램프 잠김 [SOL]
AND NOT   M12243	// R22 H/D2 (IN52) LH 그리퍼 클램프 잠김확인
OR LOAD
LOAD      M12275	// R22 H/D2 LH 그리퍼 클램프 풀림 [SOL]
AND NOT   M12244	// R22 H/D2 (IN53) LH 그리퍼 클램프 풀림확인
OR LOAD
LOAD      T2911	// R22 HD2 LH 그리퍼 클램프 이상
AND NOT   M00004	// OP1 이상해제
AND NOT   M0000C	// OP2 이상해제
OR LOAD
AND NOT   M00030	// OP LINE Emergency Stop
AND NOT   T2915	// R22 HD2 에어이상
AND NOT   T0055	// 라인1라인 메인에어 압력저하 이상
TON       T2911 100	// R22 HD2 LH 그리퍼 클램프 이상

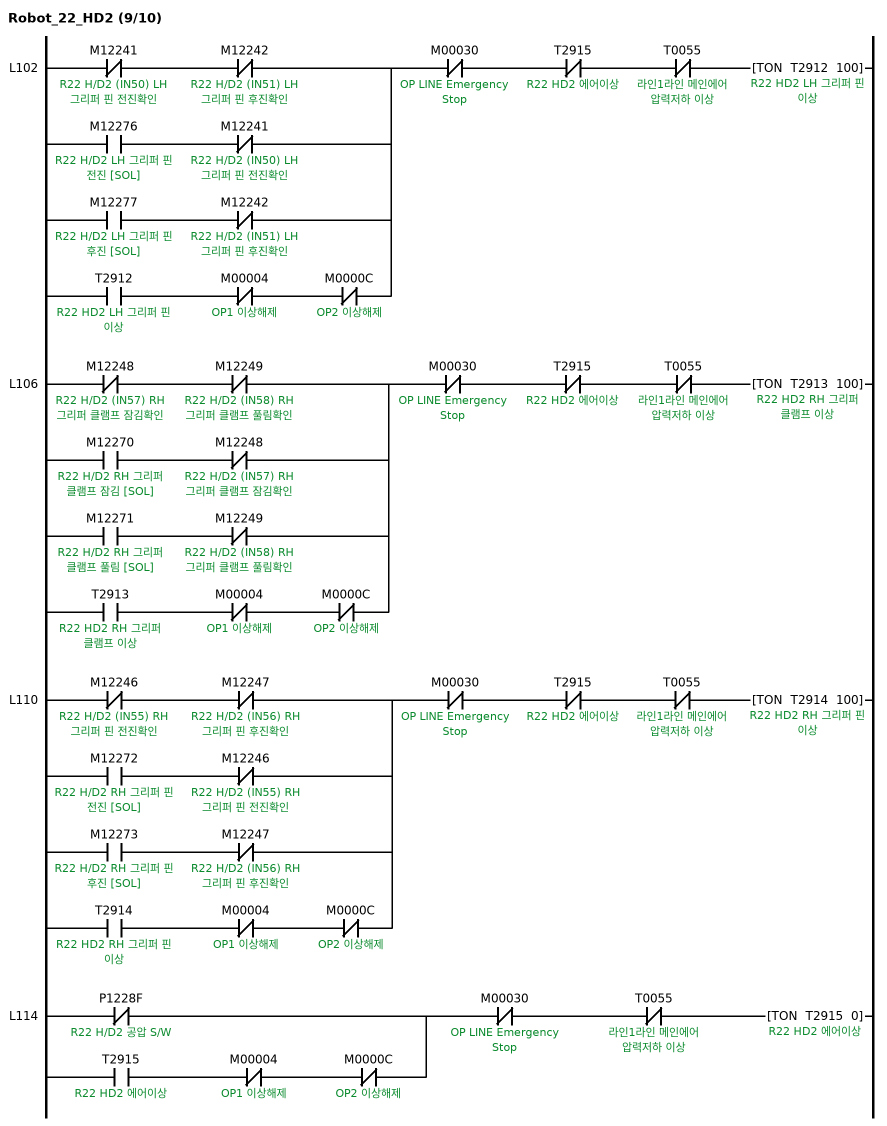
; L102
LOAD NOT  M12241	// R22 H/D2 (IN50) LH 그리퍼 핀 전진확인
AND NOT   M12242	// R22 H/D2 (IN51) LH 그리퍼 핀 후진확인
LOAD      M12276	// R22 H/D2 LH 그리퍼 핀 전진 [SOL]
AND NOT   M12241	// R22 H/D2 (IN50) LH 그리퍼 핀 전진확인
OR LOAD
LOAD      M12277	// R22 H/D2 LH 그리퍼 핀 후진 [SOL]
AND NOT   M12242	// R22 H/D2 (IN51) LH 그리퍼 핀 후진확인
OR LOAD
LOAD      T2912	// R22 HD2 LH 그리퍼 핀 이상
AND NOT   M00004	// OP1 이상해제
AND NOT   M0000C	// OP2 이상해제
OR LOAD
AND NOT   M00030	// OP LINE Emergency Stop
AND NOT   T2915	// R22 HD2 에어이상
AND NOT   T0055	// 라인1라인 메인에어 압력저하 이상
TON       T2912 100	// R22 HD2 LH 그리퍼 핀 이상
; L106
LOAD NOT  M12248	// R22 H/D2 (IN57) RH 그리퍼 클램프 잠김확인
AND NOT   M12249	// R22 H/D2 (IN58) RH 그리퍼 클램프 풀림확인
LOAD      M12270	// R22 H/D2 RH 그리퍼 클램프 잠김 [SOL]
AND NOT   M12248	// R22 H/D2 (IN57) RH 그리퍼 클램프 잠김확인
OR LOAD
LOAD      M12271	// R22 H/D2 RH 그리퍼 클램프 풀림 [SOL]
AND NOT   M12249	// R22 H/D2 (IN58) RH 그리퍼 클램프 풀림확인
OR LOAD
LOAD      T2913	// R22 HD2 RH 그리퍼 클램프 이상
AND NOT   M00004	// OP1 이상해제
AND NOT   M0000C	// OP2 이상해제
OR LOAD
AND NOT   M00030	// OP LINE Emergency Stop
AND NOT   T2915	// R22 HD2 에어이상
AND NOT   T0055	// 라인1라인 메인에어 압력저하 이상
TON       T2913 100	// R22 HD2 RH 그리퍼 클램프 이상
; L110
LOAD NOT  M12246	// R22 H/D2 (IN55) RH 그리퍼 핀 전진확인
AND NOT   M12247	// R22 H/D2 (IN56) RH 그리퍼 핀 후진확인
LOAD      M12272	// R22 H/D2 RH 그리퍼 핀 전진 [SOL]
AND NOT   M12246	// R22 H/D2 (IN55) RH 그리퍼 핀 전진확인
OR LOAD
LOAD      M12273	// R22 H/D2 RH 그리퍼 핀 후진 [SOL]
AND NOT   M12247	// R22 H/D2 (IN56) RH 그리퍼 핀 후진확인
OR LOAD
LOAD      T2914	// R22 HD2 RH 그리퍼 핀 이상
AND NOT   M00004	// OP1 이상해제
AND NOT   M0000C	// OP2 이상해제
OR LOAD
AND NOT   M00030	// OP LINE Emergency Stop
AND NOT   T2915	// R22 HD2 에어이상
AND NOT   T0055	// 라인1라인 메인에어 압력저하 이상
TON       T2914 100	// R22 HD2 RH 그리퍼 핀 이상
; L114
LOAD NOT  P1228F	// R22 H/D2 공압 S/W
LOAD      T2915	// R22 HD2 에어이상
AND NOT   M00004	// OP1 이상해제
AND NOT   M0000C	// OP2 이상해제
OR LOAD
AND NOT   M00030	// OP LINE Emergency Stop
AND NOT   T0055	// 라인1라인 메인에어 압력저하 이상
TON       T2915 0	// R22 HD2 에어이상

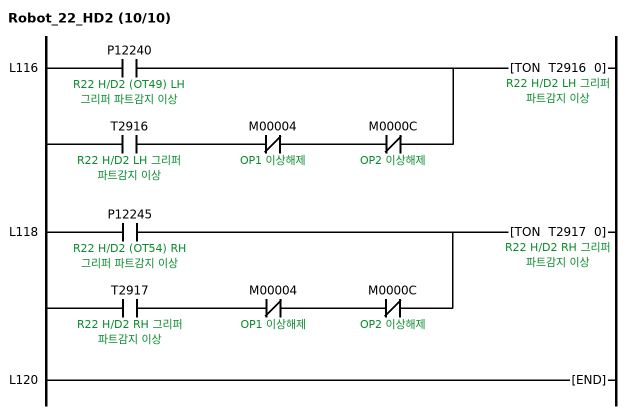
; L116
LOAD      P12240	// R22 H/D2 (OT49) LH 그리퍼 파트감지 이상
LOAD      T2916	// R22 H/D2 LH 그리퍼 파트감지 이상
AND NOT   M00004	// OP1 이상해제
AND NOT   M0000C	// OP2 이상해제
OR LOAD
TON       T2916 0	// R22 H/D2 LH 그리퍼 파트감지 이상
; L118
LOAD      P12245	// R22 H/D2 (OT54) RH 그리퍼 파트감지 이상
LOAD      T2917	// R22 H/D2 RH 그리퍼 파트감지 이상
AND NOT   M00004	// OP1 이상해제
AND NOT   M0000C	// OP2 이상해제
OR LOAD
TON       T2917 0	// R22 H/D2 RH 그리퍼 파트감지 이상
; L120
END

PROGRAM Robot_23_HD3 (task: 스캔 프로그램)

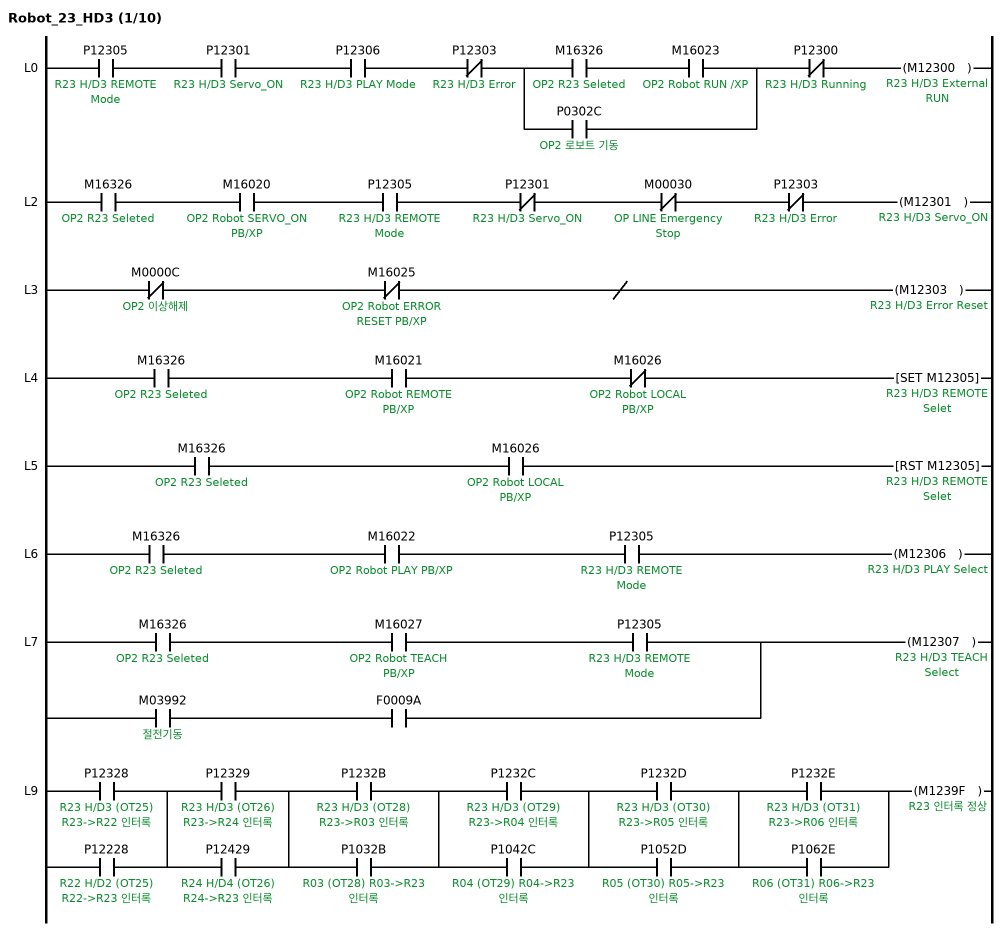
; L0
LOAD      P12305	// R23 H/D3 REMOTE Mode
AND       P12301	// R23 H/D3 Servo_ON
AND       P12306	// R23 H/D3 PLAY Mode
AND NOT   P12303	// R23 H/D3 Error
LOAD      M16326	// OP2 R23 Seleted
AND       M16023	// OP2 Robot RUN /XP
OR        P0302C	// OP2 로보트 기동
AND LOAD
AND NOT   P12300	// R23 H/D3 Running
OUT       M12300	// R23 H/D3 External RUN
; L2
LOAD      M16326	// OP2 R23 Seleted
AND       M16020	// OP2 Robot SERVO_ON PB/XP
AND       P12305	// R23 H/D3 REMOTE Mode
AND NOT   P12301	// R23 H/D3 Servo_ON
AND NOT   M00030	// OP LINE Emergency Stop
AND NOT   P12303	// R23 H/D3 Error
OUT       M12301	// R23 H/D3 Servo_ON
; L3
LOAD NOT  M0000C	// OP2 이상해제
AND NOT   M16025	// OP2 Robot ERROR RESET PB/XP
NOT
OUT       M12303	// R23 H/D3 Error Reset
; L4
LOAD      M16326	// OP2 R23 Seleted
AND       M16021	// OP2 Robot REMOTE PB/XP
AND NOT   M16026	// OP2 Robot LOCAL PB/XP
SET       M12305	// R23 H/D3 REMOTE Selet
; L5
LOAD      M16326	// OP2 R23 Seleted
AND       M16026	// OP2 Robot LOCAL PB/XP
RST       M12305	// R23 H/D3 REMOTE Selet
; L6
LOAD      M16326	// OP2 R23 Seleted
AND       M16022	// OP2 Robot PLAY PB/XP
AND       P12305	// R23 H/D3 REMOTE Mode
OUT       M12306	// R23 H/D3 PLAY Select
; L7
LOAD      M16326	// OP2 R23 Seleted
AND       M16027	// OP2 Robot TEACH PB/XP
AND       P12305	// R23 H/D3 REMOTE Mode
LOAD      M03992	// 절전기동
AND       F0009A
OR LOAD
OUT       M12307	// R23 H/D3 TEACH Select
; L9
LOAD      P12328	// R23 H/D3 (OT25) R23->R22 인터록
OR        P12228	// R22 H/D2 (OT25) R22->R23 인터록
LOAD      P12329	// R23 H/D3 (OT26) R23->R24 인터록
OR        P12429	// R24 H/D4 (OT26) R24->R23 인터록
AND LOAD
LOAD      P1232B	// R23 H/D3 (OT28) R23->R03 인터록
OR        P1032B	// R03 (OT28) R03->R23 인터록
AND LOAD
LOAD      P1232C	// R23 H/D3 (OT29) R23->R04 인터록
OR        P1042C	// R04 (OT29) R04->R23 인터록
AND LOAD
LOAD      P1232D	// R23 H/D3 (OT30) R23->R05 인터록
OR        P1052D	// R05 (OT30) R05->R23 인터록
AND LOAD
LOAD      P1232E	// R23 H/D3 (OT31) R23->R06 인터록
OR        P1062E	// R06 (OT31) R06->R23 인터록
AND LOAD
OUT       M1239F	// R23 인터록 정상

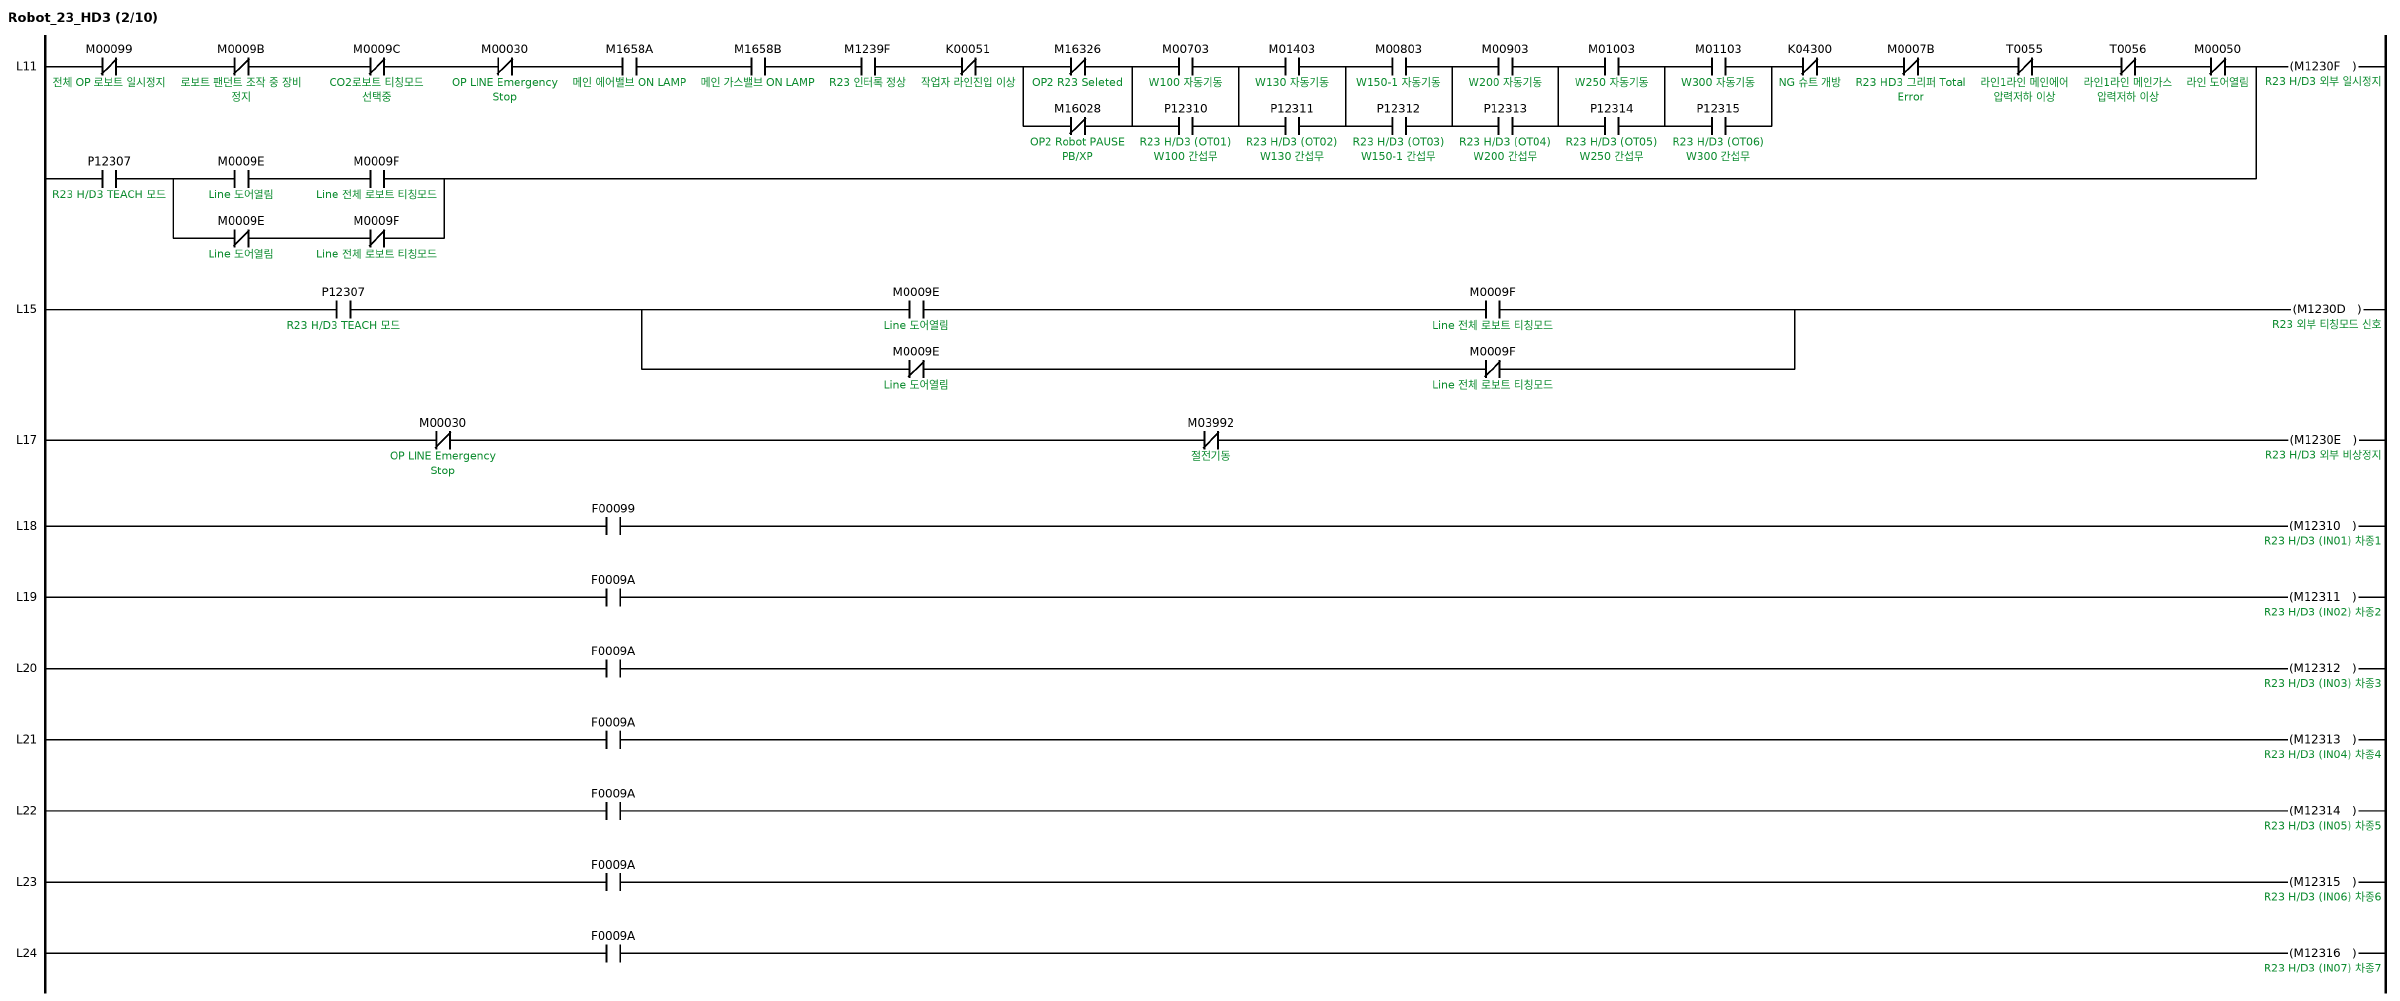
; L11
LOAD NOT  M00099	// 전체 OP 로보트 일시정지
AND NOT   M0009B	// 로보트 팬던트 조작 중 장비 정지
AND NOT   M0009C	// CO2로보트 티칭모드 선택중
AND NOT   M00030	// OP LINE Emergency Stop
AND       M1658A	// 메인 에어밸브 ON LAMP
AND       M1658B	// 메인 가스밸브 ON LAMP
AND       M1239F	// R23 인터록 정상
AND NOT   K00051	//  작업자 라인진입 이상
LOAD NOT  M16326	// OP2 R23 Seleted
OR NOT    M16028	// OP2 Robot PAUSE PB/XP
AND LOAD
LOAD      M00703	// W100 자동기동
OR        P12310	// R23 H/D3 (OT01) W100 간섭무
AND LOAD
LOAD      M01403	// W130 자동기동
OR        P12311	// R23 H/D3 (OT02) W130 간섭무
AND LOAD
LOAD      M00803	// W150-1 자동기동
OR        P12312	// R23 H/D3 (OT03) W150-1 간섭무
AND LOAD
LOAD      M00903	// W200 자동기동
OR        P12313	// R23 H/D3 (OT04) W200 간섭무
AND LOAD
LOAD      M01003	// W250 자동기동
OR        P12314	// R23 H/D3 (OT05) W250 간섭무
AND LOAD
LOAD      M01103	// W300 자동기동
OR        P12315	// R23 H/D3 (OT06) W300 간섭무
AND LOAD
AND NOT   K04300	// NG 슈트 개방
AND NOT   M0007B	// R23 HD3 그리퍼 Total Error 
AND NOT   T0055	// 라인1라인 메인에어 압력저하 이상
AND NOT   T0056	// 라인1라인 메인가스 압력저하 이상
AND NOT   M00050	// 라인 도어열림
LOAD      P12307	// R23 H/D3 TEACH 모드
LOAD      M0009E	// Line 도어열림
AND       M0009F	// Line 전체 로보트 티칭모드
LOAD NOT  M0009E	// Line 도어열림
AND NOT   M0009F	// Line 전체 로보트 티칭모드
OR LOAD
AND LOAD
OR LOAD
OUT       M1230F	// R23 H/D3 외부 일시정지
; L15
LOAD      P12307	// R23 H/D3 TEACH 모드
LOAD      M0009E	// Line 도어열림
AND       M0009F	// Line 전체 로보트 티칭모드
LOAD NOT  M0009E	// Line 도어열림
AND NOT   M0009F	// Line 전체 로보트 티칭모드
OR LOAD
AND LOAD
OUT       M1230D	// R23 외부 티칭모드 신호
; L17
LOAD NOT  M00030	// OP LINE Emergency Stop
AND NOT   M03992	// 절전기동
OUT       M1230E	// R23 H/D3 외부 비상정지 
; L18
LOAD      F00099
OUT       M12310	// R23 H/D3 (IN01) 차종1
; L19
LOAD      F0009A
OUT       M12311	// R23 H/D3 (IN02) 차종2
; L20
LOAD      F0009A
OUT       M12312	// R23 H/D3 (IN03) 차종3
; L21
LOAD      F0009A
OUT       M12313	// R23 H/D3 (IN04) 차종4
; L22
LOAD      F0009A
OUT       M12314	// R23 H/D3 (IN05) 차종5
; L23
LOAD      F0009A
OUT       M12315	// R23 H/D3 (IN06) 차종6
; L24
LOAD      F0009A
OUT       M12316	// R23 H/D3 (IN07) 차종7

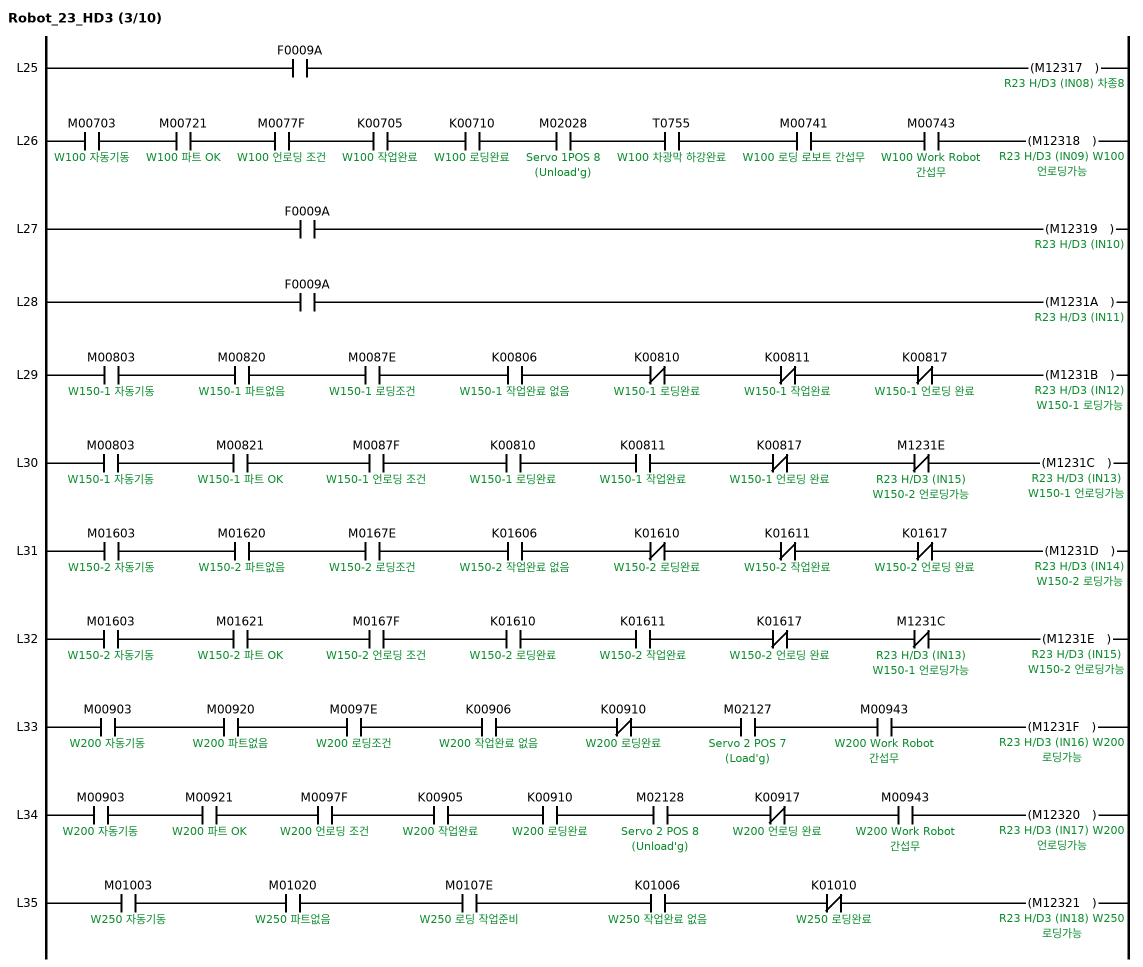
; L25
LOAD      F0009A
OUT       M12317	// R23 H/D3 (IN08) 차종8
; L26
LOAD      M00703	// W100 자동기동
AND       M00721	// W100 파트 OK
AND       M0077F	// W100 언로딩 조건
AND       K00705	// W100 작업완료
AND       K00710	// W100 로딩완료
AND       M02028	// Servo 1POS 8 (Unload'g)
AND       T0755	// W100 차광막 하강완료
AND       M00741	// W100 로딩 로보트 간섭무
AND       M00743	// W100 Work Robot 간섭무
OUT       M12318	// R23 H/D3 (IN09) W100 언로딩가능
; L27
LOAD      F0009A
OUT       M12319	// R23 H/D3 (IN10)
; L28
LOAD      F0009A
OUT       M1231A	// R23 H/D3 (IN11)
; L29
LOAD      M00803	// W150-1 자동기동
AND       M00820	// W150-1 파트없음
AND       M0087E	// W150-1 로딩조건
AND       K00806	// W150-1 작업완료 없음
AND NOT   K00810	// W150-1 로딩완료
AND NOT   K00811	// W150-1 작업완료
AND NOT   K00817	// W150-1 언로딩 완료
OUT       M1231B	// R23 H/D3 (IN12) W150-1 로딩가능
; L30
LOAD      M00803	// W150-1 자동기동
AND       M00821	// W150-1 파트 OK
AND       M0087F	// W150-1 언로딩 조건
AND       K00810	// W150-1 로딩완료
AND       K00811	// W150-1 작업완료
AND NOT   K00817	// W150-1 언로딩 완료
AND NOT   M1231E	// R23 H/D3 (IN15) W150-2 언로딩가능
OUT       M1231C	// R23 H/D3 (IN13) W150-1 언로딩가능
; L31
LOAD      M01603	// W150-2 자동기동
AND       M01620	// W150-2 파트없음
AND       M0167E	// W150-2 로딩조건
AND       K01606	// W150-2 작업완료 없음
AND NOT   K01610	// W150-2 로딩완료
AND NOT   K01611	// W150-2 작업완료
AND NOT   K01617	// W150-2 언로딩 완료
OUT       M1231D	// R23 H/D3 (IN14) W150-2 로딩가능
; L32
LOAD      M01603	// W150-2 자동기동
AND       M01621	// W150-2 파트 OK
AND       M0167F	// W150-2 언로딩 조건
AND       K01610	// W150-2 로딩완료
AND       K01611	// W150-2 작업완료
AND NOT   K01617	// W150-2 언로딩 완료
AND NOT   M1231C	// R23 H/D3 (IN13) W150-1 언로딩가능
OUT       M1231E	// R23 H/D3 (IN15) W150-2 언로딩가능
; L33
LOAD      M00903	// W200 자동기동
AND       M00920	// W200 파트없음
AND       M0097E	// W200 로딩조건
AND       K00906	// W200 작업완료 없음
AND NOT   K00910	// W200 로딩완료
AND       M02127	// Servo 2 POS 7 (Load'g)
AND       M00943	// W200 Work Robot 간섭무
OUT       M1231F	// R23 H/D3 (IN16) W200 로딩가능
; L34
LOAD      M00903	// W200 자동기동
AND       M00921	// W200 파트 OK
AND       M0097F	// W200 언로딩 조건
AND       K00905	// W200 작업완료
AND       K00910	// W200 로딩완료
AND       M02128	// Servo 2 POS 8 (Unload'g)
AND NOT   K00917	// W200 언로딩 완료
AND       M00943	// W200 Work Robot 간섭무
OUT       M12320	// R23 H/D3 (IN17) W200 언로딩가능
; L35
LOAD      M01003	// W250 자동기동
AND       M01020	// W250 파트없음
AND       M0107E	// W250 로딩 작업준비
AND       K01006	// W250 작업완료 없음
AND NOT   K01010	// W250 로딩완료
OUT       M12321	// R23 H/D3 (IN18) W250 로딩가능

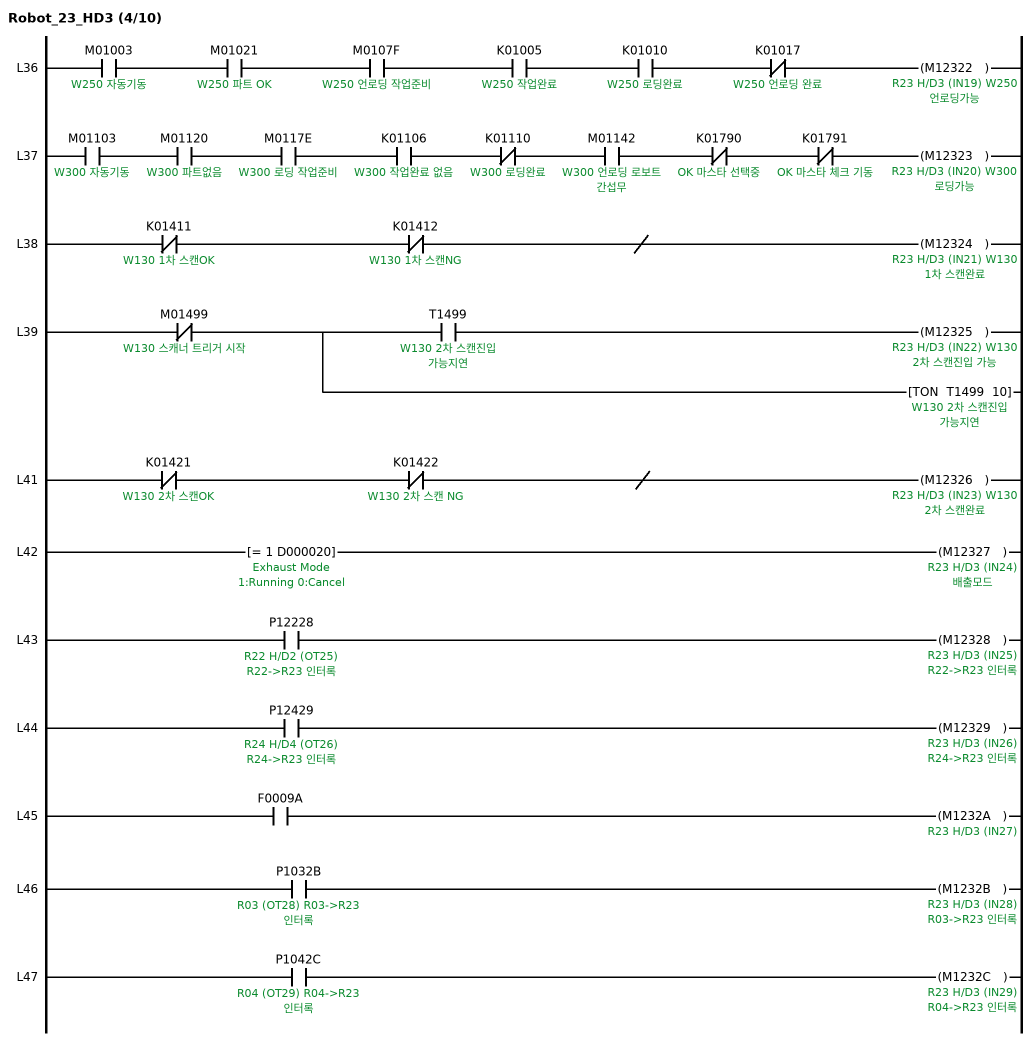
; L36
LOAD      M01003	// W250 자동기동
AND       M01021	// W250 파트 OK
AND       M0107F	// W250 언로딩 작업준비
AND       K01005	// W250 작업완료
AND       K01010	// W250 로딩완료
AND NOT   K01017	// W250 언로딩 완료
OUT       M12322	// R23 H/D3 (IN19) W250 언로딩가능
; L37
LOAD      M01103	// W300 자동기동
AND       M01120	// W300 파트없음
AND       M0117E	// W300 로딩 작업준비
AND       K01106	// W300 작업완료 없음
AND NOT   K01110	// W300 로딩완료
AND       M01142	// W300 언로딩 로보트 간섭무
AND NOT   K01790	// OK 마스타 선택중
AND NOT   K01791	// OK 마스타 체크 기동
OUT       M12323	// R23 H/D3 (IN20) W300 로딩가능
; L38
LOAD NOT  K01411	// W130 1차 스캔OK
AND NOT   K01412	// W130 1차 스캔NG
NOT
OUT       M12324	// R23 H/D3 (IN21) W130 1차 스캔완료
; L39
LOAD NOT  M01499	// W130 스캐너 트리거 시작
MPUSH
AND       T1499	// W130 2차 스캔진입 가능지연
OUT       M12325	// R23 H/D3 (IN22) W130 2차 스캔진입 가능
MPOP
TON       T1499 10	// W130 2차 스캔진입 가능지연
; L41
LOAD NOT  K01421	// W130 2차 스캔OK
AND NOT   K01422	// W130 2차 스캔 NG
NOT
OUT       M12326	// R23 H/D3 (IN23) W130 2차 스캔완료
; L42
LOAD=     1 D000020	// Exhaust Mode 1:Running 0:Cancel
OUT       M12327	// R23 H/D3 (IN24) 배출모드
; L43
LOAD      P12228	// R22 H/D2 (OT25) R22->R23 인터록
OUT       M12328	// R23 H/D3 (IN25) R22->R23 인터록
; L44
LOAD      P12429	// R24 H/D4 (OT26) R24->R23 인터록
OUT       M12329	// R23 H/D3 (IN26) R24->R23 인터록
; L45
LOAD      F0009A
OUT       M1232A	// R23 H/D3 (IN27)
; L46
LOAD      P1032B	// R03 (OT28) R03->R23 인터록
OUT       M1232B	// R23 H/D3 (IN28) R03->R23 인터록
; L47
LOAD      P1042C	// R04 (OT29) R04->R23 인터록
OUT       M1232C	// R23 H/D3 (IN29) R04->R23 인터록

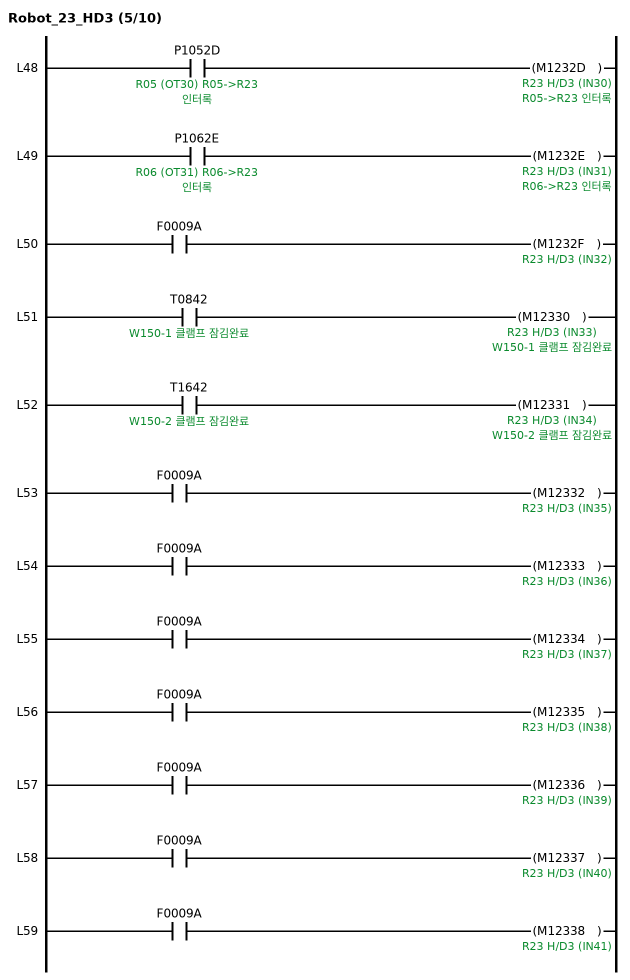
; L48
LOAD      P1052D	// R05 (OT30) R05->R23 인터록
OUT       M1232D	// R23 H/D3 (IN30) R05->R23 인터록
; L49
LOAD      P1062E	// R06 (OT31) R06->R23 인터록
OUT       M1232E	// R23 H/D3 (IN31) R06->R23 인터록
; L50
LOAD      F0009A
OUT       M1232F	// R23 H/D3 (IN32)
; L51
LOAD      T0842	// W150-1 클램프 잠김완료
OUT       M12330	// R23 H/D3 (IN33) W150-1 클램프 잠김완료
; L52
LOAD      T1642	// W150-2 클램프 잠김완료
OUT       M12331	// R23 H/D3 (IN34) W150-2 클램프 잠김완료
; L53
LOAD      F0009A
OUT       M12332	// R23 H/D3 (IN35)
; L54
LOAD      F0009A
OUT       M12333	// R23 H/D3 (IN36)
; L55
LOAD      F0009A
OUT       M12334	// R23 H/D3 (IN37)
; L56
LOAD      F0009A
OUT       M12335	// R23 H/D3 (IN38)
; L57
LOAD      F0009A
OUT       M12336	// R23 H/D3 (IN39)
; L58
LOAD      F0009A
OUT       M12337	// R23 H/D3 (IN40)
; L59
LOAD      F0009A
OUT       M12338	// R23 H/D3 (IN41)

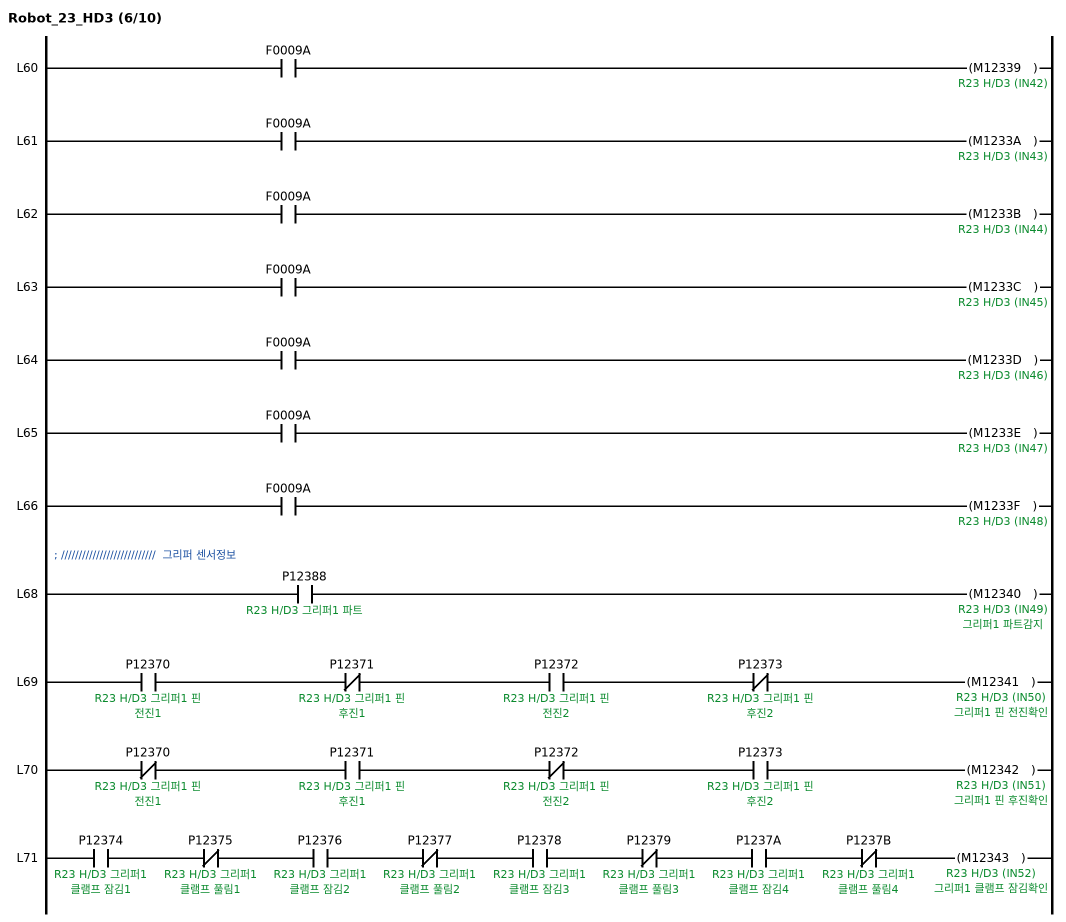
; L60
LOAD      F0009A
OUT       M12339	// R23 H/D3 (IN42)
; L61
LOAD      F0009A
OUT       M1233A	// R23 H/D3 (IN43)
; L62
LOAD      F0009A
OUT       M1233B	// R23 H/D3 (IN44)
; L63
LOAD      F0009A
OUT       M1233C	// R23 H/D3 (IN45)
; L64
LOAD      F0009A
OUT       M1233D	// R23 H/D3 (IN46)
; L65
LOAD      F0009A
OUT       M1233E	// R23 H/D3 (IN47)
; L66
LOAD      F0009A
OUT       M1233F	// R23 H/D3 (IN48)
// ///////////////////////////  그리퍼 센서정보
; L68
LOAD      P12388	// R23 H/D3 그리퍼1 파트
OUT       M12340	// R23 H/D3 (IN49) 그리퍼1 파트감지
; L69
LOAD      P12370	// R23 H/D3 그리퍼1 핀 전진1
AND NOT   P12371	// R23 H/D3 그리퍼1 핀 후진1
AND       P12372	// R23 H/D3 그리퍼1 핀 전진2
AND NOT   P12373	// R23 H/D3 그리퍼1 핀 후진2
OUT       M12341	// R23 H/D3 (IN50) 그리퍼1 핀 전진확인
; L70
LOAD NOT  P12370	// R23 H/D3 그리퍼1 핀 전진1
AND       P12371	// R23 H/D3 그리퍼1 핀 후진1
AND NOT   P12372	// R23 H/D3 그리퍼1 핀 전진2
AND       P12373	// R23 H/D3 그리퍼1 핀 후진2
OUT       M12342	// R23 H/D3 (IN51) 그리퍼1 핀 후진확인
; L71
LOAD      P12374	// R23 H/D3 그리퍼1 클램프 잠김1
AND NOT   P12375	// R23 H/D3 그리퍼1 클램프 풀림1
AND       P12376	// R23 H/D3 그리퍼1 클램프 잠김2
AND NOT   P12377	// R23 H/D3 그리퍼1 클램프 풀림2
AND       P12378	// R23 H/D3 그리퍼1 클램프 잠김3
AND NOT   P12379	// R23 H/D3 그리퍼1 클램프 풀림3
AND       P1237A	// R23 H/D3 그리퍼1 클램프 잠김4
AND NOT   P1237B	// R23 H/D3 그리퍼1 클램프 풀림4
OUT       M12343	// R23 H/D3 (IN52) 그리퍼1 클램프 잠김확인

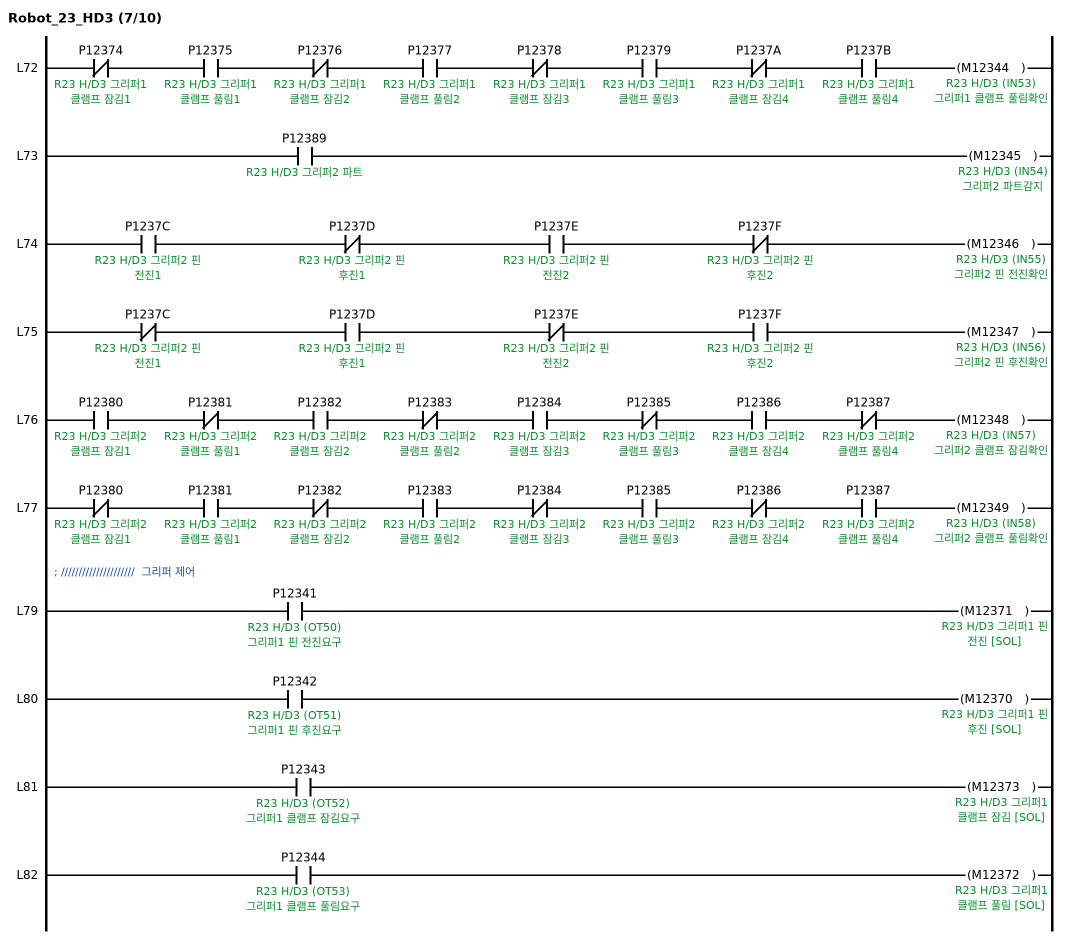
; L72
LOAD NOT  P12374	// R23 H/D3 그리퍼1 클램프 잠김1
AND       P12375	// R23 H/D3 그리퍼1 클램프 풀림1
AND NOT   P12376	// R23 H/D3 그리퍼1 클램프 잠김2
AND       P12377	// R23 H/D3 그리퍼1 클램프 풀림2
AND NOT   P12378	// R23 H/D3 그리퍼1 클램프 잠김3
AND       P12379	// R23 H/D3 그리퍼1 클램프 풀림3
AND NOT   P1237A	// R23 H/D3 그리퍼1 클램프 잠김4
AND       P1237B	// R23 H/D3 그리퍼1 클램프 풀림4
OUT       M12344	// R23 H/D3 (IN53) 그리퍼1 클램프 풀림확인
; L73
LOAD      P12389	// R23 H/D3 그리퍼2 파트
OUT       M12345	// R23 H/D3 (IN54) 그리퍼2 파트감지
; L74
LOAD      P1237C	// R23 H/D3 그리퍼2 핀 전진1
AND NOT   P1237D	// R23 H/D3 그리퍼2 핀 후진1
AND       P1237E	// R23 H/D3 그리퍼2 핀 전진2
AND NOT   P1237F	// R23 H/D3 그리퍼2 핀 후진2
OUT       M12346	// R23 H/D3 (IN55) 그리퍼2 핀 전진확인
; L75
LOAD NOT  P1237C	// R23 H/D3 그리퍼2 핀 전진1
AND       P1237D	// R23 H/D3 그리퍼2 핀 후진1
AND NOT   P1237E	// R23 H/D3 그리퍼2 핀 전진2
AND       P1237F	// R23 H/D3 그리퍼2 핀 후진2
OUT       M12347	// R23 H/D3 (IN56) 그리퍼2 핀 후진확인
; L76
LOAD      P12380	// R23 H/D3 그리퍼2 클램프 잠김1
AND NOT   P12381	// R23 H/D3 그리퍼2 클램프 풀림1
AND       P12382	// R23 H/D3 그리퍼2 클램프 잠김2
AND NOT   P12383	// R23 H/D3 그리퍼2 클램프 풀림2
AND       P12384	// R23 H/D3 그리퍼2 클램프 잠김3
AND NOT   P12385	// R23 H/D3 그리퍼2 클램프 풀림3
AND       P12386	// R23 H/D3 그리퍼2 클램프 잠김4
AND NOT   P12387	// R23 H/D3 그리퍼2 클램프 풀림4
OUT       M12348	// R23 H/D3 (IN57) 그리퍼2 클램프 잠김확인
; L77
LOAD NOT  P12380	// R23 H/D3 그리퍼2 클램프 잠김1
AND       P12381	// R23 H/D3 그리퍼2 클램프 풀림1
AND NOT   P12382	// R23 H/D3 그리퍼2 클램프 잠김2
AND       P12383	// R23 H/D3 그리퍼2 클램프 풀림2
AND NOT   P12384	// R23 H/D3 그리퍼2 클램프 잠김3
AND       P12385	// R23 H/D3 그리퍼2 클램프 풀림3
AND NOT   P12386	// R23 H/D3 그리퍼2 클램프 잠김4
AND       P12387	// R23 H/D3 그리퍼2 클램프 풀림4
OUT       M12349	// R23 H/D3 (IN58) 그리퍼2 클램프 풀림확인
// /////////////////////  그리퍼 제어
; L79
LOAD      P12341	// R23 H/D3 (OT50) 그리퍼1 핀 전진요구
OUT       M12371	// R23 H/D3 그리퍼1 핀 전진 [SOL]
; L80
LOAD      P12342	// R23 H/D3 (OT51) 그리퍼1 핀 후진요구
OUT       M12370	// R23 H/D3 그리퍼1 핀 후진 [SOL]
; L81
LOAD      P12343	// R23 H/D3 (OT52) 그리퍼1 클램프 잠김요구
OUT       M12373	// R23 H/D3 그리퍼1 클램프 잠김 [SOL]
; L82
LOAD      P12344	// R23 H/D3 (OT53) 그리퍼1 클램프 풀림요구
OUT       M12372	// R23 H/D3 그리퍼1 클램프 풀림 [SOL]

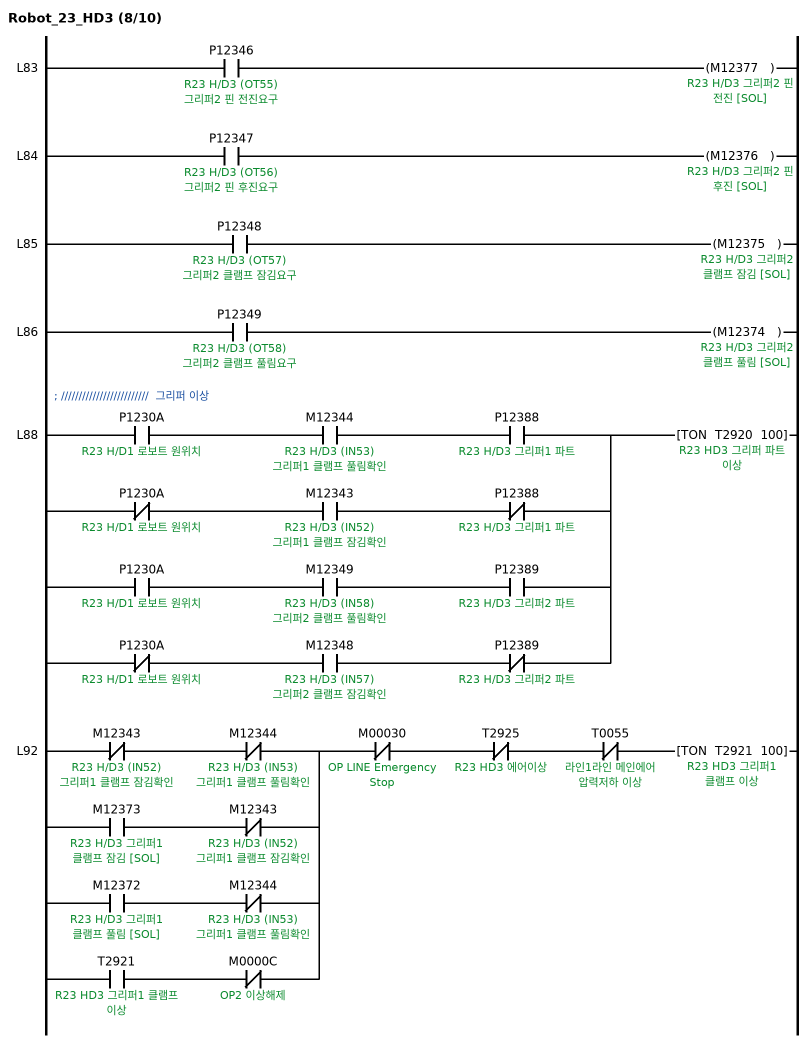
; L83
LOAD      P12346	// R23 H/D3 (OT55) 그리퍼2 핀 전진요구
OUT       M12377	// R23 H/D3 그리퍼2 핀 전진 [SOL]
; L84
LOAD      P12347	// R23 H/D3 (OT56) 그리퍼2 핀 후진요구
OUT       M12376	// R23 H/D3 그리퍼2 핀 후진 [SOL]
; L85
LOAD      P12348	// R23 H/D3 (OT57) 그리퍼2 클램프 잠김요구
OUT       M12375	// R23 H/D3 그리퍼2 클램프 잠김 [SOL]
; L86
LOAD      P12349	// R23 H/D3 (OT58) 그리퍼2 클램프 풀림요구
OUT       M12374	// R23 H/D3 그리퍼2 클램프 풀림 [SOL]
// /////////////////////////  그리퍼 이상
; L88
LOAD      P1230A	// R23 H/D1 로보트 원위치
AND       M12344	// R23 H/D3 (IN53) 그리퍼1 클램프 풀림확인
AND       P12388	// R23 H/D3 그리퍼1 파트
LOAD NOT  P1230A	// R23 H/D1 로보트 원위치
AND       M12343	// R23 H/D3 (IN52) 그리퍼1 클램프 잠김확인
AND NOT   P12388	// R23 H/D3 그리퍼1 파트
OR LOAD
LOAD      P1230A	// R23 H/D1 로보트 원위치
AND       M12349	// R23 H/D3 (IN58) 그리퍼2 클램프 풀림확인
AND       P12389	// R23 H/D3 그리퍼2 파트
OR LOAD
LOAD NOT  P1230A	// R23 H/D1 로보트 원위치
AND       M12348	// R23 H/D3 (IN57) 그리퍼2 클램프 잠김확인
AND NOT   P12389	// R23 H/D3 그리퍼2 파트
OR LOAD
TON       T2920 100	// R23 HD3 그리퍼 파트 이상
; L92
LOAD NOT  M12343	// R23 H/D3 (IN52) 그리퍼1 클램프 잠김확인
AND NOT   M12344	// R23 H/D3 (IN53) 그리퍼1 클램프 풀림확인
LOAD      M12373	// R23 H/D3 그리퍼1 클램프 잠김 [SOL]
AND NOT   M12343	// R23 H/D3 (IN52) 그리퍼1 클램프 잠김확인
OR LOAD
LOAD      M12372	// R23 H/D3 그리퍼1 클램프 풀림 [SOL]
AND NOT   M12344	// R23 H/D3 (IN53) 그리퍼1 클램프 풀림확인
OR LOAD
LOAD      T2921	// R23 HD3 그리퍼1 클램프 이상
AND NOT   M0000C	// OP2 이상해제
OR LOAD
AND NOT   M00030	// OP LINE Emergency Stop
AND NOT   T2925	// R23 HD3 에어이상
AND NOT   T0055	// 라인1라인 메인에어 압력저하 이상
TON       T2921 100	// R23 HD3 그리퍼1 클램프 이상

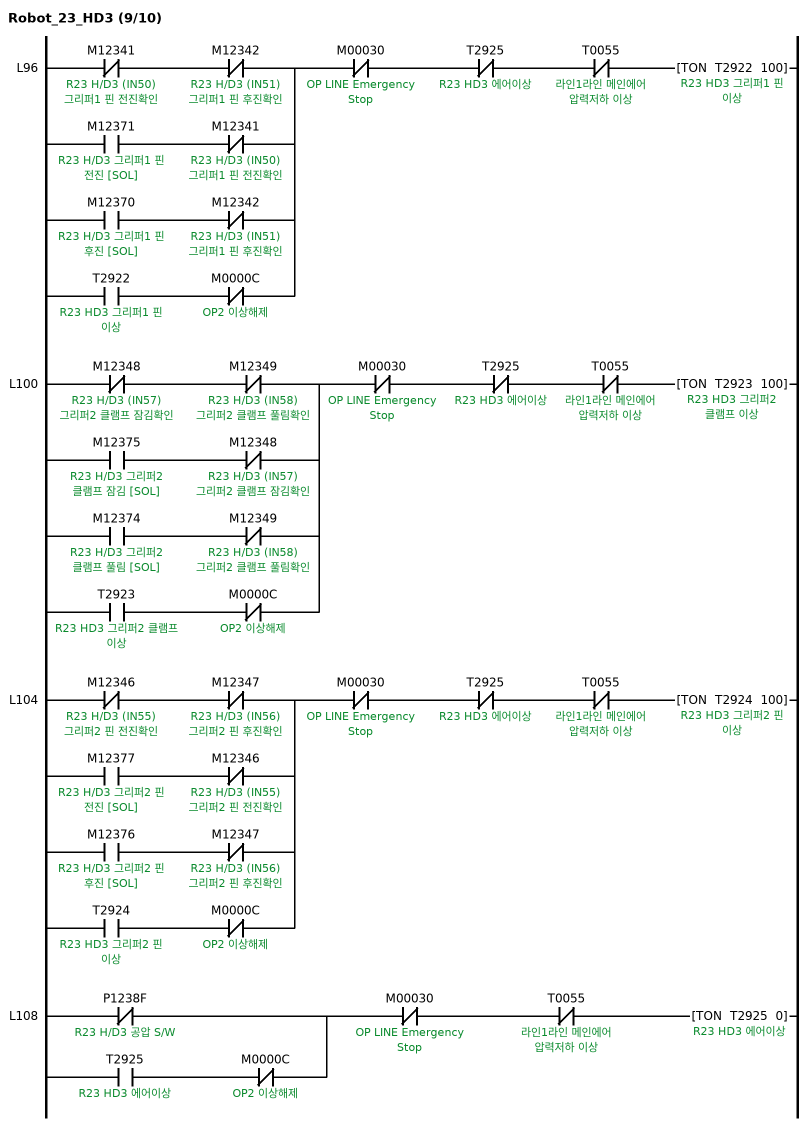
; L96
LOAD NOT  M12341	// R23 H/D3 (IN50) 그리퍼1 핀 전진확인
AND NOT   M12342	// R23 H/D3 (IN51) 그리퍼1 핀 후진확인
LOAD      M12371	// R23 H/D3 그리퍼1 핀 전진 [SOL]
AND NOT   M12341	// R23 H/D3 (IN50) 그리퍼1 핀 전진확인
OR LOAD
LOAD      M12370	// R23 H/D3 그리퍼1 핀 후진 [SOL]
AND NOT   M12342	// R23 H/D3 (IN51) 그리퍼1 핀 후진확인
OR LOAD
LOAD      T2922	// R23 HD3 그리퍼1 핀 이상
AND NOT   M0000C	// OP2 이상해제
OR LOAD
AND NOT   M00030	// OP LINE Emergency Stop
AND NOT   T2925	// R23 HD3 에어이상
AND NOT   T0055	// 라인1라인 메인에어 압력저하 이상
TON       T2922 100	// R23 HD3 그리퍼1 핀 이상
; L100
LOAD NOT  M12348	// R23 H/D3 (IN57) 그리퍼2 클램프 잠김확인
AND NOT   M12349	// R23 H/D3 (IN58) 그리퍼2 클램프 풀림확인
LOAD      M12375	// R23 H/D3 그리퍼2 클램프 잠김 [SOL]
AND NOT   M12348	// R23 H/D3 (IN57) 그리퍼2 클램프 잠김확인
OR LOAD
LOAD      M12374	// R23 H/D3 그리퍼2 클램프 풀림 [SOL]
AND NOT   M12349	// R23 H/D3 (IN58) 그리퍼2 클램프 풀림확인
OR LOAD
LOAD      T2923	// R23 HD3 그리퍼2 클램프 이상
AND NOT   M0000C	// OP2 이상해제
OR LOAD
AND NOT   M00030	// OP LINE Emergency Stop
AND NOT   T2925	// R23 HD3 에어이상
AND NOT   T0055	// 라인1라인 메인에어 압력저하 이상
TON       T2923 100	// R23 HD3 그리퍼2 클램프 이상
; L104
LOAD NOT  M12346	// R23 H/D3 (IN55) 그리퍼2 핀 전진확인
AND NOT   M12347	// R23 H/D3 (IN56) 그리퍼2 핀 후진확인
LOAD      M12377	// R23 H/D3 그리퍼2 핀 전진 [SOL]
AND NOT   M12346	// R23 H/D3 (IN55) 그리퍼2 핀 전진확인
OR LOAD
LOAD      M12376	// R23 H/D3 그리퍼2 핀 후진 [SOL]
AND NOT   M12347	// R23 H/D3 (IN56) 그리퍼2 핀 후진확인
OR LOAD
LOAD      T2924	// R23 HD3 그리퍼2 핀 이상
AND NOT   M0000C	// OP2 이상해제
OR LOAD
AND NOT   M00030	// OP LINE Emergency Stop
AND NOT   T2925	// R23 HD3 에어이상
AND NOT   T0055	// 라인1라인 메인에어 압력저하 이상
TON       T2924 100	// R23 HD3 그리퍼2 핀 이상
; L108
LOAD NOT  P1238F	// R23 H/D3 공압 S/W
LOAD      T2925	// R23 HD3 에어이상
AND NOT   M0000C	// OP2 이상해제
OR LOAD
AND NOT   M00030	// OP LINE Emergency Stop
AND NOT   T0055	// 라인1라인 메인에어 압력저하 이상
TON       T2925 0	// R23 HD3 에어이상

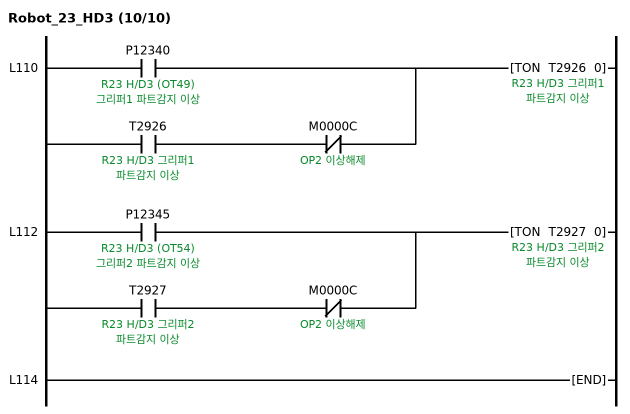
; L110
LOAD      P12340	// R23 H/D3 (OT49) 그리퍼1 파트감지 이상
LOAD      T2926	// R23 H/D3 그리퍼1 파트감지 이상
AND NOT   M0000C	// OP2 이상해제
OR LOAD
TON       T2926 0	// R23 H/D3 그리퍼1 파트감지 이상
; L112
LOAD      P12345	// R23 H/D3 (OT54) 그리퍼2 파트감지 이상
LOAD      T2927	// R23 H/D3 그리퍼2 파트감지 이상
AND NOT   M0000C	// OP2 이상해제
OR LOAD
TON       T2927 0	// R23 H/D3 그리퍼2 파트감지 이상
; L114
END

PROGRAM Robot_24_HD4 (task: 스캔 프로그램)

